LIN {X 0,Y 217.024,Z 808.035,A -85,B 0,C 180,E1 -22006.463,E2 -22006.463} C_VEL
LIN {X 0,Y 209.804,Z 820.642,A -85,B 0,C 180,E1 -22009.848,E2 -22009.848} C_VEL
LIN {X 0,Y 205.023,Z 828.704,A -85,B 0,C 180,E1 -22012.523,E2 -22012.523} C_VEL
LIN {X 0,Y 199.918,Z 836.875,A -85,B 0,C 180,E1 -22015.774,E2 -22015.774} C_VEL
LIN {X 0,Y 196.083,Z 843.017,A -85,B 0,C 180,E1 -22018.688,E2 -22018.688} C_VEL
LIN {X 0,Y 191.79,Z 849.969,A -85,B 0,C 180,E1 -22022.739,E2 -22022.739} C_VEL
LIN {X 0,Y 188.385,Z 855.734,A -85,B 0,C 180,E1 -22026.939,E2 -22026.939} C_VEL
LIN {X 0,Y 186.27,Z 859.773,A -85,B 0,C 180,E1 -22030.606,E2 -22030.606} C_VEL
LIN {X 0,Y 184.562,Z 863.22,A -85,B 0,C 180,E1 -22034.541,E2 -22034.541} C_VEL
LIN {X 0,Y 183.409,Z 866.084,A -85,B 0,C 180,E1 -22038.954,E2 -22038.954} C_VEL
LIN {X 0,Y 183.157,Z 867.229,A -85,B 0,C 180,E1 -22041.171,E2 -22041.171} C_VEL
LIN {X 0,Y 183.027,Z 868.67,A -85,B 0,C 180,E1 -22045.596,E2 -22045.596} C_VEL
LIN {X 0,Y 183.139,Z 869.152,A -85,B 0,C 180,E1 -22050,E2 -22050} C_VEL
LIN {X 0,Y 183.027,Z 868.67,A -85,B 0,C 180,E1 -22054.404,E2 -22054.404} C_VEL
LIN {X 0,Y 183.156,Z 867.229,A -85,B 0,C 180,E1 -22058.829,E2 -22058.829} C_VEL
LIN {X 0,Y 183.829,Z 864.826,A -85,B 0,C 180,E1 -22063.261,E2 -22063.261} C_VEL
LIN {X 0,Y 185.438,Z 861.443,A -85,B 0,C 180,E1 -22067.649,E2 -22067.649} C_VEL
LIN {X 0,Y 187.698,Z 857.024,A -85,B 0,C 180,E1 -22071.989,E2 -22071.989} C_VEL
LIN {X 0,Y 190.882,Z 851.516,A -85,B 0,C 180,E1 -22076.22,E2 -22076.22} C_VEL
LIN {X 0,Y 194.222,Z 845.918,A -85,B 0,C 180,E1 -22079.721,E2 -22079.721} C_VEL
LIN {X 0,Y 198.584,Z 838.981,A -85,B 0,C 180,E1 -22083.267,E2 -22083.267} C_VEL
LIN {X 0,Y 202.834,Z 832.332,A -85,B 0,C 180,E1 -22086.087,E2 -22086.087} C_VEL
LIN {X 0,Y 207.695,Z 824.178,A -85,B 0,C 180,E1 -22089.026,E2 -22089.026} C_VEL
LIN {X 0,Y 212.368,Z 816.196,A -85,B 0,C 180,E1 -22091.441,E2 -22091.441} C_VEL
LIN {X 0,Y 217.847,Z 806.411,A -85,B 0,C 180,E1 -22093.916,E2 -22093.916} C_VEL
LIN {X 0,Y 223.353,Z 796.062,A -85,B 0,C 180,E1 -22096.079,E2 -22096.079} C_VEL
LIN {X 0,Y 228.421,Z 785.635,A -85,B 0,C 180,E1 -22097.924,E2 -22097.924} C_VEL
LIN {X 0,Y 233.261,Z 774.829,A -85,B 0,C 180,E1 -22099.53,E2 -22099.53} C_VEL
LIN {X 0,Y 237.755,Z 763.897,A -85,B 0,C 180,E1 -22100.889,E2 -22100.889} C_VEL
LIN {X 0,Y 242.076,Z 752.106,A -85,B 0,C 180,E1 -22102.121,E2 -22102.121} C_VEL
LIN {X 0,Y 246.197,Z 739.235,A -85,B 0,C 180,E1 -22103.231,E2 -22103.231} C_VEL
LIN {X 0,Y 249.836,Z 726.035,A -85,B 0,C 180,E1 -22104.144,E2 -22104.144} C_VEL
LIN {X 0,Y 252.794,Z 713.298,A -85,B 0,C 180,E1 -22104.836,E2 -22104.836} C_VEL
LIN {X 0,Y 255.143,Z 700.698,A -85,B 0,C 180,E1 -22105.376,E2 -22105.376} C_VEL
LIN {X 0,Y 256.972,Z 687.246,A -85,B 0,C 180,E1 -22105.822,E2 -22105.822} C_VEL
LIN {X 0,Y 259.606,Z 655.333,A -85,B 0,C 180,E1 -22106.613,E2 -22106.613} C_VEL
LIN {X 0,Y 264.674,Z 589.177,A -85,B 0,C 180,E1 -22108.172,E2 -22108.172} C_VEL
LIN {X 0,Y 260.374,Z 578.709,A -85,B 0,C 180,E1 -22110.28,E2 -22110.28} C_VEL
LIN {X 0,Y 255.377,Z 567.773,A -85,B 0,C 180,E1 -22112.939,E2 -22112.939} C_VEL
LIN {X 0,Y 251.472,Z 560.216,A -85,B 0,C 180,E1 -22115.215,E2 -22115.215} C_VEL
LIN {X 0,Y 247.589,Z 554.194,A -85,B 0,C 180,E1 -22117.66,E2 -22117.66} C_VEL
LIN {X 0,Y 245.205,Z 550.628,A -85,B 0,C 180,E1 -22119.327,E2 -22119.327} C_VEL
LIN {X 0,Y 242.508,Z 546.779,A -85,B 0,C 180,E1 -22121.41,E2 -22121.41} C_VEL
LIN {X 0,Y 239.491,Z 542.43,A -85,B 0,C 180,E1 -22124.116,E2 -22124.116} C_VEL
LIN {X 0,Y 237.073,Z 538.972,A -85,B 0,C 180,E1 -22126.718,E2 -22126.718} C_VEL
LIN {X 0,Y 236.559,Z 538.249,A -85,B 0,C 180,E1 -22127.343,E2 -22127.343} C_VEL
LIN {X 0,Y 234.058,Z 535.194,A -85,B 0,C 180,E1 -22130.93,E2 -22130.93} C_VEL
LIN {X 0,Y 233.366,Z 533.383,A -85,B 0,C 180,E1 -22132.429,E2 -22132.429} C_VEL
LIN {X 0,Y 231.434,Z 531.641,A -85,B 0,C 180,E1 -22140,E2 -22140} C_VEL
LIN {X 0,Y 233.419,Z 533.525,A -85,B 0,C 180,E1 -22148.113,E2 -22148.113} C_VEL
LIN {X 0,Y 235.107,Z 536.867,A -85,B 0,C 180,E1 -22151.204,E2 -22151.204} C_VEL
LIN {X 0,Y 237.005,Z 538.845,A -85,B 0,C 180,E1 -22153.613,E2 -22153.613} C_VEL
LIN {X 0,Y 239.475,Z 542.534,A -85,B 0,C 180,E1 -22156.298,E2 -22156.298} C_VEL
LIN {X 0,Y 240.592,Z 544.125,A -85,B 0,C 180,E1 -22157.353,E2 -22157.353} C_VEL
LIN {X 0,Y 243.915,Z 548.714,A -85,B 0,C 180,E1 -22160.118,E2 -22160.118} C_VEL
LIN {X 0,Y 246.909,Z 553.171,A -85,B 0,C 180,E1 -22162.296,E2 -22162.296} C_VEL
LIN {X 0,Y 251.503,Z 560.18,A -85,B 0,C 180,E1 -22165.214,E2 -22165.214} C_VEL
LIN {X 0,Y 256.264,Z 567.994,A -85,B 0,C 180,E1 -22167.872,E2 -22167.872} C_VEL
LIN {X 0,Y 263.831,Z 578.938,A -85,B 0,C 180,E1 -22171.427,E2 -22171.427} C_VEL
LIN {X 0,Y 270.208,Z 586.445,A -85,B 0,C 180,E1 -22173.945,E2 -22173.945} C_VEL
LIN {X 0,Y 277.709,Z 593.975,A -85,B 0,C 180,E1 -22176.52,E2 -22176.52} C_VEL
LIN {X 0,Y 287.772,Z 602.451,A -85,B 0,C 180,E1 -22179.509,E2 -22179.509} C_VEL
LIN {X 0,Y 295.037,Z 608.473,A -85,B 0,C 180,E1 -22181.667,E2 -22181.667} C_VEL
LIN {X 0,Y 301.973,Z 614.367,A -85,B 0,C 180,E1 -22183.92,E2 -22183.92} C_VEL
LIN {X 0,Y 307.887,Z 619.394,A -85,B 0,C 180,E1 -22185.977,E2 -22185.977} C_VEL
LIN {X 0,Y 314.535,Z 625.112,A -85,B 0,C 180,E1 -22188.552,E2 -22188.552} C_VEL
LIN {X 0,Y 320.194,Z 630.065,A -85,B 0,C 180,E1 -22190.886,E2 -22190.886} C_VEL
LIN {X 0,Y 327.166,Z 636.13,A -85,B 0,C 180,E1 -22193.896,E2 -22193.896} C_VEL
LIN {X 0,Y 331.947,Z 639.962,A -85,B 0,C 180,E1 -22196.053,E2 -22196.053} C_VEL
LIN {X 0,Y 336.603,Z 643.968,A -85,B 0,C 180,E1 -22198.269,E2 -22198.269} C_VEL
LIN {X 0,Y 340.503,Z 647.021,A -85,B 0,C 180,E1 -22200.202,E2 -22200.202} C_VEL
LIN {X 0,Y 344.944,Z 651.021,A -85,B 0,C 180,E1 -22202.581,E2 -22202.581} C_VEL
LIN {X 0,Y 349.886,Z 654.477,A -85,B 0,C 180,E1 -22205.377,E2 -22205.377} C_VEL
LIN {X 0,Y 353.537,Z 657.803,A -85,B 0,C 180,E1 -22207.688,E2 -22207.688} C_VEL
LIN {X 0,Y 357.378,Z 660.485,A -85,B 0,C 180,E1 -22210.301,E2 -22210.301} C_VEL
LIN {X 0,Y 359.995,Z 662.174,A -85,B 0,C 180,E1 -22212.302,E2 -22212.302} C_VEL
LIN {X 0,Y 362.803,Z 664.895,A -85,B 0,C 180,E1 -22214.773,E2 -22214.773} C_VEL
LIN {X 0,Y 365.298,Z 666.919,A -85,B 0,C 180,E1 -22217.353,E2 -22217.353} C_VEL
LIN {X 0,Y 367.182,Z 668.028,A -85,B 0,C 180,E1 -22219.57,E2 -22219.57} C_VEL
LIN {X 0,Y 369.013,Z 668.858,A -85,B 0,C 180,E1 -22222.339,E2 -22222.339} C_VEL
LIN {X 0,Y 370.309,Z 669.612,A -85,B 0,C 180,E1 -22225.096,E2 -22225.096} C_VEL
LIN {X 0,Y 371.028,Z 669.847,A -85,B 0,C 180,E1 -22227.829,E2 -22227.829} C_VEL
LIN {X 0,Y 371.228,Z 669.986,A -85,B 0,C 180,E1 -22230,E2 -22230} C_VEL
LIN {X 0,Y 371.028,Z 669.845,A -85,B 0,C 180,E1 -22232.171,E2 -22232.171} C_VEL
LIN {X 0,Y 370.309,Z 669.617,A -85,B 0,C 180,E1 -22234.904,E2 -22234.904} C_VEL
LIN {X 0,Y 369.013,Z 668.859,A -85,B 0,C 180,E1 -22237.661,E2 -22237.661} C_VEL
LIN {X 0,Y 367.28,Z 668.119,A -85,B 0,C 180,E1 -22240.312,E2 -22240.312} C_VEL
LIN {X 0,Y 364.987,Z 666.71,A -85,B 0,C 180,E1 -22243,E2 -22243} C_VEL
LIN {X 0,Y 362.396,Z 664.592,A -85,B 0,C 180,E1 -22245.579,E2 -22245.579} C_VEL
LIN {X 0,Y 359.357,Z 661.588,A -85,B 0,C 180,E1 -22248.235,E2 -22248.235} C_VEL
LIN {X 0,Y 356.069,Z 659.663,A -85,B 0,C 180,E1 -22250.596,E2 -22250.596} C_VEL
LIN {X 0,Y 352.093,Z 656.652,A -85,B 0,C 180,E1 -22253.233,E2 -22253.233} C_VEL
LIN {X 0,Y 348.854,Z 653.633,A -85,B 0,C 180,E1 -22255.248,E2 -22255.248} C_VEL
LIN {X 0,Y 344.683,Z 650.803,A -85,B 0,C 180,E1 -22257.562,E2 -22257.562} C_VEL
LIN {X 0,Y 339.913,Z 646.465,A -85,B 0,C 180,E1 -22260.097,E2 -22260.097} C_VEL
LIN {X 0,Y 334.266,Z 642.131,A -85,B 0,C 180,E1 -22262.846,E2 -22262.846} C_VEL
LIN {X 0,Y 329.785,Z 638.132,A -85,B 0,C 180,E1 -22264.941,E2 -22264.941} C_VEL
LIN {X 0,Y 324.302,Z 633.671,A -85,B 0,C 180,E1 -22267.357,E2 -22267.357} C_VEL
LIN {X 0,Y 319.804,Z 629.722,A -85,B 0,C 180,E1 -22269.277,E2 -22269.277} C_VEL
LIN {X 0,Y 314.166,Z 624.78,A -85,B 0,C 180,E1 -22271.598,E2 -22271.598} C_VEL
LIN {X 0,Y 307.596,Z 619.166,A -85,B 0,C 180,E1 -22274.126,E2 -22274.126} C_VEL
LIN {X 0,Y 301.98,Z 614.344,A -85,B 0,C 180,E1 -22276.079,E2 -22276.079} C_VEL
LIN {X 0,Y 295.594,Z 608.892,A -85,B 0,C 180,E1 -22278.155,E2 -22278.155} C_VEL
LIN {X 0,Y 288.716,Z 603.223,A -85,B 0,C 180,E1 -22280.223,E2 -22280.223} C_VEL
LIN {X 0,Y 279.821,Z 595.822,A -85,B 0,C 180,E1 -22282.818,E2 -22282.818} C_VEL
LIN {X 0,Y 271.936,Z 588.351,A -85,B 0,C 180,E1 -22285.426,E2 -22285.426} C_VEL
LIN {X 0,Y 264.195,Z 579.408,A -85,B 0,C 180,E1 -22288.419,E2 -22288.419} C_VEL
LIN {X 0,Y 256.457,Z 568.307,A -85,B 0,C 180,E1 -22292.027,E2 -22292.027} C_VEL
LIN {X 0,Y 251.912,Z 560.875,A -85,B 0,C 180,E1 -22294.542,E2 -22294.542} C_VEL
LIN {X 0,Y 247.439,Z 553.984,A -85,B 0,C 180,E1 -22297.343,E2 -22297.343} C_VEL
LIN {X 0,Y 244.959,Z 550.237,A -85,B 0,C 180,E1 -22299.094,E2 -22299.094} C_VEL
LIN {X 0,Y 242.778,Z 547.152,A -85,B 0,C 180,E1 -22300.775,E2 -22300.775} C_VEL
LIN {X 0,Y 239.641,Z 542.684,A -85,B 0,C 180,E1 -22303.55,E2 -22303.55} C_VEL
LIN {X 0,Y 237.165,Z 539.221,A -85,B 0,C 180,E1 -22306.178,E2 -22306.178} C_VEL
LIN {X 0,Y 236.484,Z 538.21,A -85,B 0,C 180,E1 -22307.012,E2 -22307.012} C_VEL
LIN {X 0,Y 234.186,Z 535.427,A -85,B 0,C 180,E1 -22310.282,E2 -22310.282} C_VEL
LIN {X 0,Y 233.268,Z 533.307,A -85,B 0,C 180,E1 -22312.208,E2 -22312.208} C_VEL
LIN {X 0,Y 231.434,Z 531.64,A -85,B 0,C 180,E1 -22320,E2 -22320} C_VEL
LIN {X 0,Y 233.413,Z 533.486,A -85,B 0,C 180,E1 -22327.679,E2 -22327.679} C_VEL
LIN {X 0,Y 235.097,Z 536.825,A -85,B 0,C 180,E1 -22330.769,E2 -22330.769} C_VEL
LIN {X 0,Y 236.992,Z 538.793,A -85,B 0,C 180,E1 -22333.178,E2 -22333.178} C_VEL
LIN {X 0,Y 239.142,Z 542.101,A -85,B 0,C 180,E1 -22335.556,E2 -22335.556} C_VEL
LIN {X 0,Y 240.394,Z 543.725,A -85,B 0,C 180,E1 -22336.744,E2 -22336.744} C_VEL
LIN {X 0,Y 243.948,Z 548.807,A -85,B 0,C 180,E1 -22339.732,E2 -22339.732} C_VEL
LIN {X 0,Y 246.984,Z 553.277,A -85,B 0,C 180,E1 -22341.93,E2 -22341.93} C_VEL
LIN {X 0,Y 251.076,Z 559.526,A -85,B 0,C 180,E1 -22344.544,E2 -22344.544} C_VEL
LIN {X 0,Y 254.166,Z 565.218,A -85,B 0,C 180,E1 -22346.369,E2 -22346.369} C_VEL
LIN {X 0,Y 259.878,Z 577.475,A -85,B 0,C 180,E1 -22349.463,E2 -22349.463} C_VEL
LIN {X 0,Y 264.683,Z 589.177,A -85,B 0,C 180,E1 -22351.831,E2 -22351.831} C_VEL
LIN {X 0,Y 257.13,Z 685.944,A -85,B 0,C 180,E1 -22354.143,E2 -22354.143} C_VEL
LIN {X 0,Y 255.437,Z 698.699,A -85,B 0,C 180,E1 -22354.546,E2 -22354.546} C_VEL
LIN {X 0,Y 253.09,Z 711.765,A -85,B 0,C 180,E1 -22355.086,E2 -22355.086} C_VEL
LIN {X 0,Y 250.427,Z 723.566,A -85,B 0,C 180,E1 -22355.7,E2 -22355.7} C_VEL
LIN {X 0,Y 247.095,Z 736.159,A -85,B 0,C 180,E1 -22356.536,E2 -22356.536} C_VEL
LIN {X 0,Y 243.326,Z 748.397,A -85,B 0,C 180,E1 -22357.538,E2 -22357.538} C_VEL
LIN {X 0,Y 238.912,Z 760.899,A -85,B 0,C 180,E1 -22358.783,E2 -22358.783} C_VEL
LIN {X 0,Y 234.406,Z 772.222,A -85,B 0,C 180,E1 -22360.135,E2 -22360.135} C_VEL
LIN {X 0,Y 229.479,Z 783.349,A -85,B 0,C 180,E1 -22361.713,E2 -22361.713} C_VEL
LIN {X 0,Y 224.821,Z 793.183,A -85,B 0,C 180,E1 -22363.384,E2 -22363.384} C_VEL
LIN {X 0,Y 219.863,Z 802.865,A -85,B 0,C 180,E1 -22365.314,E2 -22365.314} C_VEL
LIN {X 0,Y 217.024,Z 808.035,A -85,B 0,C 180,E1 -22366.463,E2 -22366.463} C_VEL
LIN {X 0,Y 214.287,Z 812.154,A -85,B 0,C 180,E1 -22367.329,E2 -22367.329} C_VEL
LIN {X 0,Y 208.286,Z 818.645,A -85,B 0,C 180,E1 -22368.566,E2 -22368.566} C_VEL
LIN {X 0,Y 202.265,Z 824.691,A -85,B 0,C 180,E1 -22369.975,E2 -22369.975} C_VEL
LIN {X 0,Y 199.551,Z 828.11,A -85,B 0,C 180,E1 -22371.106,E2 -22371.106} C_VEL
LIN {X 0,Y 193.984,Z 836.662,A -85,B 0,C 180,E1 -22374.573,E2 -22374.573} C_VEL
LIN {X 0,Y 189.938,Z 842.803,A -85,B 0,C 180,E1 -22377.554,E2 -22377.554} C_VEL
LIN {X 0,Y 185.391,Z 849.755,A -85,B 0,C 180,E1 -22381.715,E2 -22381.715} C_VEL
LIN {X 0,Y 181.771,Z 855.521,A -85,B 0,C 180,E1 -22386.049,E2 -22386.049} C_VEL
LIN {X 0,Y 179.735,Z 859.145,A -85,B 0,C 180,E1 -22389.396,E2 -22389.396} C_VEL
LIN {X 0,Y 177.65,Z 863.008,A -85,B 0,C 180,E1 -22393.924,E2 -22393.924} C_VEL
LIN {X 0,Y 176.388,Z 865.873,A -85,B 0,C 180,E1 -22398.509,E2 -22398.509} C_VEL
LIN {X 0,Y 176.08,Z 867.017,A -85,B 0,C 180,E1 -22400.813,E2 -22400.813} C_VEL
LIN {X 0,Y 175.936,Z 868.459,A -85,B 0,C 180,E1 -22405.418,E2 -22405.418} C_VEL
LIN {X 0,Y 176.048,Z 868.943,A -85,B 0,C 180,E1 -22410,E2 -22410} C_VEL
LIN {X 0,Y 175.936,Z 868.459,A -85,B 0,C 180,E1 -22414.582,E2 -22414.582} C_VEL
LIN {X 0,Y 176.079,Z 867.017,A -85,B 0,C 180,E1 -22419.187,E2 -22419.187} C_VEL
LIN {X 0,Y 176.855,Z 864.614,A -85,B 0,C 180,E1 -22423.794,E2 -22423.794} C_VEL
LIN {X 0,Y 179.323,Z 859.848,A -85,B 0,C 180,E1 -22429.847,E2 -22429.847} C_VEL
LIN {X 0,Y 181.033,Z 856.811,A -85,B 0,C 180,E1 -22432.843,E2 -22432.843} C_VEL
LIN {X 0,Y 184.415,Z 851.302,A -85,B 0,C 180,E1 -22437.213,E2 -22437.213} C_VEL
LIN {X 0,Y 187.644,Z 846.219,A -85,B 0,C 180,E1 -22440.521,E2 -22440.521} C_VEL
LIN {X 0,Y 192.602,Z 838.768,A -85,B 0,C 180,E1 -22444.442,E2 -22444.442} C_VEL
LIN {X 0,Y 197.05,Z 832.119,A -85,B 0,C 180,E1 -22447.323,E2 -22447.323} C_VEL
LIN {X 0,Y 201.93,Z 824.313,A -85,B 0,C 180,E1 -22450.2,E2 -22450.2} C_VEL
LIN {X 0,Y 207.021,Z 815.983,A -85,B 0,C 180,E1 -22452.761,E2 -22452.761} C_VEL
LIN {X 0,Y 212.732,Z 806.198,A -85,B 0,C 180,E1 -22455.257,E2 -22455.257} C_VEL
LIN {X 0,Y 217.992,Z 796.721,A -85,B 0,C 180,E1 -22457.266,E2 -22457.266} C_VEL
LIN {X 0,Y 223.141,Z 786.567,A -85,B 0,C 180,E1 -22459.102,E2 -22459.102} C_VEL
LIN {X 0,Y 228.685,Z 774.618,A -85,B 0,C 180,E1 -22460.893,E2 -22460.893} C_VEL
LIN {X 0,Y 233.303,Z 763.685,A -85,B 0,C 180,E1 -22462.254,E2 -22462.254} C_VEL
LIN {X 0,Y 237.693,Z 752.113,A -85,B 0,C 180,E1 -22463.457,E2 -22463.457} C_VEL
LIN {X 0,Y 241.996,Z 739.024,A -85,B 0,C 180,E1 -22464.584,E2 -22464.584} C_VEL
LIN {X 0,Y 245.739,Z 725.825,A -85,B 0,C 180,E1 -22465.487,E2 -22465.487} C_VEL
LIN {X 0,Y 248.78,Z 713.088,A -85,B 0,C 180,E1 -22466.171,E2 -22466.171} C_VEL
LIN {X 0,Y 251.178,Z 700.488,A -85,B 0,C 180,E1 -22466.708,E2 -22466.708} C_VEL
LIN {X 0,Y 253.054,Z 687.036,A -85,B 0,C 180,E1 -22467.151,E2 -22467.151} C_VEL
LIN {X 0,Y 255.611,Z 656.913,A -85,B 0,C 180,E1 -22467.905,E2 -22467.905} C_VEL
LIN {X 0,Y 260.741,Z 592.077,A -85,B 0,C 180,E1 -22469.427,E2 -22469.427} C_VEL
LIN {X 0,Y 256.898,Z 582.594,A -85,B 0,C 180,E1 -22471.433,E2 -22471.433} C_VEL
LIN {X 0,Y 252.212,Z 572.078,A -85,B 0,C 180,E1 -22474.095,E2 -22474.095} C_VEL
LIN {X 0,Y 249.051,Z 565.842,A -85,B 0,C 180,E1 -22476.047,E2 -22476.047} C_VEL
LIN {X 0,Y 244.194,Z 558.051,A -85,B 0,C 180,E1 -22479.349,E2 -22479.349} C_VEL
LIN {X 0,Y 240.903,Z 553.362,A -85,B 0,C 180,E1 -22481.942,E2 -22481.942} C_VEL
LIN {X 0,Y 238.071,Z 549.141,A -85,B 0,C 180,E1 -22484.592,E2 -22484.592} C_VEL
LIN {X 0,Y 235.63,Z 545.389,A -85,B 0,C 180,E1 -22487.375,E2 -22487.375} C_VEL
LIN {X 0,Y 232.899,Z 541.908,A -85,B 0,C 180,E1 -22491.431,E2 -22491.431} C_VEL
LIN {X 0,Y 232.289,Z 540.323,A -85,B 0,C 180,E1 -22492.83,E2 -22492.83} C_VEL
LIN {X 0,Y 230.568,Z 538.691,A -85,B 0,C 180,E1 -22500,E2 -22500} C_VEL
LIN {X 0,Y 232.394,Z 540.489,A -85,B 0,C 180,E1 -22507.821,E2 -22507.821} C_VEL
LIN {X 0,Y 234.094,Z 543.891,A -85,B 0,C 180,E1 -22511.034,E2 -22511.034} C_VEL
LIN {X 0,Y 235.74,Z 545.661,A -85,B 0,C 180,E1 -22513.194,E2 -22513.194} C_VEL
LIN {X 0,Y 238.295,Z 549.47,A -85,B 0,C 180,E1 -22516.051,E2 -22516.051} C_VEL
LIN {X 0,Y 242.459,Z 555.551,A -85,B 0,C 180,E1 -22519.747,E2 -22519.747} C_VEL
LIN {X 0,Y 245.212,Z 559.806,A -85,B 0,C 180,E1 -22521.82,E2 -22521.82} C_VEL
LIN {X 0,Y 249.252,Z 566.131,A -85,B 0,C 180,E1 -22524.492,E2 -22524.492} C_VEL
LIN {X 0,Y 253.711,Z 573.674,A -85,B 0,C 180,E1 -22527.102,E2 -22527.102} C_VEL
LIN {X 0,Y 261.405,Z 585.093,A -85,B 0,C 180,E1 -22530.865,E2 -22530.865} C_VEL
LIN {X 0,Y 267.642,Z 592.574,A -85,B 0,C 180,E1 -22533.409,E2 -22533.409} C_VEL
LIN {X 0,Y 275.276,Z 600.336,A -85,B 0,C 180,E1 -22536.103,E2 -22536.103} C_VEL
LIN {X 0,Y 289.9,Z 612.757,A -85,B 0,C 180,E1 -22540.475,E2 -22540.475} C_VEL
LIN {X 0,Y 296.185,Z 617.8,A -85,B 0,C 180,E1 -22542.391,E2 -22542.391} C_VEL
LIN {X 0,Y 302.458,Z 622.865,A -85,B 0,C 180,E1 -22544.429,E2 -22544.429} C_VEL
LIN {X 0,Y 308.854,Z 628.471,A -85,B 0,C 180,E1 -22546.732,E2 -22546.732} C_VEL
LIN {X 0,Y 313.492,Z 632.478,A -85,B 0,C 180,E1 -22548.54,E2 -22548.54} C_VEL
LIN {X 0,Y 319.336,Z 637.404,A -85,B 0,C 180,E1 -22550.94,E2 -22550.94} C_VEL
LIN {X 0,Y 325.614,Z 642.904,A -85,B 0,C 180,E1 -22553.642,E2 -22553.642} C_VEL
LIN {X 0,Y 330.476,Z 646.77,A -85,B 0,C 180,E1 -22555.815,E2 -22555.815} C_VEL
LIN {X 0,Y 335.102,Z 650.715,A -85,B 0,C 180,E1 -22557.99,E2 -22557.99} C_VEL
LIN {X 0,Y 338.902,Z 653.671,A -85,B 0,C 180,E1 -22559.871,E2 -22559.871} C_VEL
LIN {X 0,Y 343.55,Z 657.813,A -85,B 0,C 180,E1 -22562.326,E2 -22562.326} C_VEL
LIN {X 0,Y 348.565,Z 661.301,A -85,B 0,C 180,E1 -22565.136,E2 -22565.136} C_VEL
LIN {X 0,Y 352.247,Z 664.636,A -85,B 0,C 180,E1 -22567.427,E2 -22567.427} C_VEL
LIN {X 0,Y 356.173,Z 667.387,A -85,B 0,C 180,E1 -22570.095,E2 -22570.095} C_VEL
LIN {X 0,Y 358.955,Z 669.162,A -85,B 0,C 180,E1 -22572.175,E2 -22572.175} C_VEL
LIN {X 0,Y 361.661,Z 671.815,A -85,B 0,C 180,E1 -22574.557,E2 -22574.557} C_VEL
LIN {X 0,Y 364.213,Z 673.832,A -85,B 0,C 180,E1 -22577.117,E2 -22577.117} C_VEL
LIN {X 0,Y 366.284,Z 675.068,A -85,B 0,C 180,E1 -22579.544,E2 -22579.544} C_VEL
LIN {X 0,Y 368.135,Z 675.877,A -85,B 0,C 180,E1 -22582.32,E2 -22582.32} C_VEL
LIN {X 0,Y 369.44,Z 676.657,A -85,B 0,C 180,E1 -22585.084,E2 -22585.084} C_VEL
LIN {X 0,Y 370.159,Z 676.892,A -85,B 0,C 180,E1 -22587.824,E2 -22587.824} C_VEL
LIN {X 0,Y 370.363,Z 677.032,A -85,B 0,C 180,E1 -22590,E2 -22590} C_VEL
LIN {X 0,Y 370.159,Z 676.891,A -85,B 0,C 180,E1 -22592.176,E2 -22592.176} C_VEL
LIN {X 0,Y 369.439,Z 676.663,A -85,B 0,C 180,E1 -22594.915,E2 -22594.915} C_VEL
LIN {X 0,Y 368.134,Z 675.885,A -85,B 0,C 180,E1 -22597.68,E2 -22597.68} C_VEL
LIN {X 0,Y 366.382,Z 675.159,A -85,B 0,C 180,E1 -22600.338,E2 -22600.338} C_VEL
LIN {X 0,Y 364.085,Z 673.731,A -85,B 0,C 180,E1 -22603.033,E2 -22603.033} C_VEL
LIN {X 0,Y 361.459,Z 671.656,A -85,B 0,C 180,E1 -22605.62,E2 -22605.62} C_VEL
LIN {X 0,Y 358.395,Z 668.607,A -85,B 0,C 180,E1 -22608.285,E2 -22608.285} C_VEL
LIN {X 0,Y 355.091,Z 666.685,A -85,B 0,C 180,E1 -22610.656,E2 -22610.656} C_VEL
LIN {X 0,Y 351.069,Z 663.714,A -85,B 0,C 180,E1 -22613.303,E2 -22613.303} C_VEL
LIN {X 0,Y 347.314,Z 660.308,A -85,B 0,C 180,E1 -22615.608,E2 -22615.608} C_VEL
LIN {X 0,Y 343.32,Z 657.597,A -85,B 0,C 180,E1 -22617.803,E2 -22617.803} C_VEL
LIN {X 0,Y 338.616,Z 653.421,A -85,B 0,C 180,E1 -22620.274,E2 -22620.274} C_VEL
LIN {X 0,Y 332.904,Z 649.018,A -85,B 0,C 180,E1 -22623.043,E2 -22623.043} C_VEL
LIN {X 0,Y 327.743,Z 644.483,A -85,B 0,C 180,E1 -22625.428,E2 -22625.428} C_VEL
LIN {X 0,Y 322.376,Z 640.13,A -85,B 0,C 180,E1 -22627.769,E2 -22627.769} C_VEL
LIN {X 0,Y 317.673,Z 636.043,A -85,B 0,C 180,E1 -22629.749,E2 -22629.749} C_VEL
LIN {X 0,Y 312.278,Z 631.353,A -85,B 0,C 180,E1 -22631.947,E2 -22631.947} C_VEL
LIN {X 0,Y 305.786,Z 625.92,A -85,B 0,C 180,E1 -22634.382,E2 -22634.382} C_VEL
LIN {X 0,Y 300.757,Z 621.582,A -85,B 0,C 180,E1 -22636.124,E2 -22636.124} C_VEL
LIN {X 0,Y 294.652,Z 616.46,A -85,B 0,C 180,E1 -22638.099,E2 -22638.099} C_VEL
LIN {X 0,Y 286.82,Z 610.155,A -85,B 0,C 180,E1 -22640.426,E2 -22640.426} C_VEL
LIN {X 0,Y 276.881,Z 601.705,A -85,B 0,C 180,E1 -22643.381,E2 -22643.381} C_VEL
LIN {X 0,Y 269.548,Z 594.713,A -85,B 0,C 180,E1 -22645.877,E2 -22645.877} C_VEL
LIN {X 0,Y 261.638,Z 585.413,A -85,B 0,C 180,E1 -22649.032,E2 -22649.032} C_VEL
LIN {X 0,Y 253.855,Z 573.918,A -85,B 0,C 180,E1 -22652.82,E2 -22652.82} C_VEL
LIN {X 0,Y 248.762,Z 565.295,A -85,B 0,C 180,E1 -22655.818,E2 -22655.818} C_VEL
LIN {X 0,Y 243.681,Z 557.331,A -85,B 0,C 180,E1 -22659.311,E2 -22659.311} C_VEL
LIN {X 0,Y 241.172,Z 553.688,A -85,B 0,C 180,E1 -22661.304,E2 -22661.304} C_VEL
LIN {X 0,Y 238.084,Z 549.235,A -85,B 0,C 180,E1 -22664.155,E2 -22664.155} C_VEL
LIN {X 0,Y 235.68,Z 545.544,A -85,B 0,C 180,E1 -22666.885,E2 -22666.885} C_VEL
LIN {X 0,Y 233.021,Z 542.13,A -85,B 0,C 180,E1 -22670.78,E2 -22670.78} C_VEL
LIN {X 0,Y 232.196,Z 540.262,A -85,B 0,C 180,E1 -22672.61,E2 -22672.61} C_VEL
LIN {X 0,Y 230.568,Z 538.689,A -85,B 0,C 180,E1 -22680,E2 -22680} C_VEL
LIN {X 0,Y 232.418,Z 540.568,A -85,B 0,C 180,E1 -22687.466,E2 -22687.466} C_VEL
LIN {X 0,Y 234.156,Z 543.929,A -85,B 0,C 180,E1 -22690.703,E2 -22690.703} C_VEL
LIN {X 0,Y 235.768,Z 545.676,A -85,B 0,C 180,E1 -22692.809,E2 -22692.809} C_VEL
LIN {X 0,Y 238.175,Z 549.264,A -85,B 0,C 180,E1 -22695.511,E2 -22695.511} C_VEL
LIN {X 0,Y 242.12,Z 555.053,A -85,B 0,C 180,E1 -22699.06,E2 -22699.06} C_VEL
LIN {X 0,Y 244.964,Z 559.36,A -85,B 0,C 180,E1 -22701.222,E2 -22701.222} C_VEL
LIN {X 0,Y 249.162,Z 566.055,A -85,B 0,C 180,E1 -22704.025,E2 -22704.025} C_VEL
LIN {X 0,Y 252.103,Z 571.844,A -85,B 0,C 180,E1 -22705.84,E2 -22705.84} C_VEL
LIN {X 0,Y 257.284,Z 583.384,A -85,B 0,C 180,E1 -22708.768,E2 -22708.768} C_VEL
LIN {X 0,Y 260.754,Z 592.12,A -85,B 0,C 180,E1 -22710.579,E2 -22710.579} C_VEL
LIN {X 0,Y 253.204,Z 685.744,A -85,B 0,C 180,E1 -22712.81,E2 -22712.81} C_VEL
LIN {X 0,Y 251.316,Z 699.488,A -85,B 0,C 180,E1 -22713.249,E2 -22713.249} C_VEL
LIN {X 0,Y 248.914,Z 712.321,A -85,B 0,C 180,E1 -22713.784,E2 -22713.784} C_VEL
LIN {X 0,Y 246.034,Z 724.59,A -85,B 0,C 180,E1 -22714.432,E2 -22714.432} C_VEL
LIN {X 0,Y 242.605,Z 736.973,A -85,B 0,C 180,E1 -22715.26,E2 -22715.26} C_VEL
LIN {X 0,Y 239.2,Z 747.796,A -85,B 0,C 180,E1 -22716.152,E2 -22716.152} C_VEL
LIN {X 0,Y 235.1,Z 759.189,A -85,B 0,C 180,E1 -22717.26,E2 -22717.26} C_VEL
LIN {X 0,Y 230.424,Z 770.705,A -85,B 0,C 180,E1 -22718.597,E2 -22718.597} C_VEL
LIN {X 0,Y 225.346,Z 781.995,A -85,B 0,C 180,E1 -22720.175,E2 -22720.175} C_VEL
LIN {X 0,Y 219.961,Z 792.967,A -85,B 0,C 180,E1 -22722.026,E2 -22722.026} C_VEL
LIN {X 0,Y 214.808,Z 802.653,A -85,B 0,C 180,E1 -22723.964,E2 -22723.964} C_VEL
LIN {X 0,Y 208.882,Z 812.852,A -85,B 0,C 180,E1 -22726.392,E2 -22726.392} C_VEL
LIN {X 0,Y 203.489,Z 821.808,A -85,B 0,C 180,E1 -22728.989,E2 -22728.989} C_VEL
LIN {X 0,Y 199.551,Z 828.11,A -85,B 0,C 180,E1 -22731.106,E2 -22731.106} C_VEL
LIN {X 0,Y 196.88,Z 831.469,A -85,B 0,C 180,E1 -22732.295,E2 -22732.295} C_VEL
LIN {X 0,Y 193.446,Z 834.798,A -85,B 0,C 180,E1 -22733.363,E2 -22733.363} C_VEL
LIN {X 0,Y 185.114,Z 841.749,A -85,B 0,C 180,E1 -22735.98,E2 -22735.98} C_VEL
LIN {X 0,Y 182.584,Z 844.418,A -85,B 0,C 180,E1 -22737.401,E2 -22737.401} C_VEL
LIN {X 0,Y 179.05,Z 849.541,A -85,B 0,C 180,E1 -22740.618,E2 -22740.618} C_VEL
LIN {X 0,Y 175.191,Z 855.308,A -85,B 0,C 180,E1 -22745.089,E2 -22745.089} C_VEL
LIN {X 0,Y 172.991,Z 858.932,A -85,B 0,C 180,E1 -22748.554,E2 -22748.554} C_VEL
LIN {X 0,Y 170.745,Z 862.795,A -85,B 0,C 180,E1 -22753.255,E2 -22753.255} C_VEL
LIN {X 0,Y 169.367,Z 865.661,A -85,B 0,C 180,E1 -22758.026,E2 -22758.026} C_VEL
LIN {X 0,Y 169.027,Z 866.806,A -85,B 0,C 180,E1 -22760.426,E2 -22760.426} C_VEL
LIN {X 0,Y 168.845,Z 868.249,A -85,B 0,C 180,E1 -22765.225,E2 -22765.225} C_VEL
LIN {X 0,Y 168.959,Z 868.733,A -85,B 0,C 180,E1 -22770,E2 -22770} C_VEL
LIN {X 0,Y 168.845,Z 868.249,A -85,B 0,C 180,E1 -22774.775,E2 -22774.775} C_VEL
LIN {X 0,Y 169.025,Z 866.806,A -85,B 0,C 180,E1 -22779.574,E2 -22779.574} C_VEL
LIN {X 0,Y 169.904,Z 864.402,A -85,B 0,C 180,E1 -22784.37,E2 -22784.37} C_VEL
LIN {X 0,Y 172.371,Z 859.939,A -85,B 0,C 180,E1 -22790.319,E2 -22790.319} C_VEL
LIN {X 0,Y 174.399,Z 856.597,A -85,B 0,C 180,E1 -22793.764,E2 -22793.764} C_VEL
LIN {X 0,Y 178.017,Z 851.088,A -85,B 0,C 180,E1 -22798.277,E2 -22798.277} C_VEL
LIN {X 0,Y 181.647,Z 845.761,A -85,B 0,C 180,E1 -22801.819,E2 -22801.819} C_VEL
LIN {X 0,Y 186.703,Z 838.555,A -85,B 0,C 180,E1 -22805.693,E2 -22805.693} C_VEL
LIN {X 0,Y 191.337,Z 831.905,A -85,B 0,C 180,E1 -22808.639,E2 -22808.639} C_VEL
LIN {X 0,Y 196.32,Z 824.355,A -85,B 0,C 180,E1 -22811.471,E2 -22811.471} C_VEL
LIN {X 0,Y 201.8,Z 815.77,A -85,B 0,C 180,E1 -22814.148,E2 -22814.148} C_VEL
LIN {X 0,Y 207.75,Z 805.987,A -85,B 0,C 180,E1 -22816.661,E2 -22816.661} C_VEL
LIN {X 0,Y 212.807,Z 797.217,A -85,B 0,C 180,E1 -22818.548,E2 -22818.548} C_VEL
LIN {X 0,Y 218.504,Z 786.354,A -85,B 0,C 180,E1 -22820.527,E2 -22820.527} C_VEL
LIN {X 0,Y 224.244,Z 774.406,A -85,B 0,C 180,E1 -22822.311,E2 -22822.311} C_VEL
LIN {X 0,Y 229.011,Z 763.475,A -85,B 0,C 180,E1 -22823.664,E2 -22823.664} C_VEL
LIN {X 0,Y 233.83,Z 751.017,A -85,B 0,C 180,E1 -22824.944,E2 -22824.944} C_VEL
LIN {X 0,Y 237.931,Z 738.814,A -85,B 0,C 180,E1 -22825.985,E2 -22825.985} C_VEL
LIN {X 0,Y 241.779,Z 725.615,A -85,B 0,C 180,E1 -22826.877,E2 -22826.877} C_VEL
LIN {X 0,Y 244.903,Z 712.879,A -85,B 0,C 180,E1 -22827.549,E2 -22827.549} C_VEL
LIN {X 0,Y 247.343,Z 700.278,A -85,B 0,C 180,E1 -22828.086,E2 -22828.086} C_VEL
LIN {X 0,Y 249.26,Z 686.825,A -85,B 0,C 180,E1 -22828.527,E2 -22828.527} C_VEL
LIN {X 0,Y 252.209,Z 653.122,A -85,B 0,C 180,E1 -22829.354,E2 -22829.354} C_VEL
LIN {X 0,Y 256.922,Z 594.922,A -85,B 0,C 180,E1 -22830.73,E2 -22830.73} C_VEL
LIN {X 0,Y 252.23,Z 583.394,A -85,B 0,C 180,E1 -22833.378,E2 -22833.378} C_VEL
LIN {X 0,Y 248.359,Z 574.803,A -85,B 0,C 180,E1 -22835.783,E2 -22835.783} C_VEL
LIN {X 0,Y 246.189,Z 570.671,A -85,B 0,C 180,E1 -22837.221,E2 -22837.221} C_VEL
LIN {X 0,Y 241.853,Z 563.699,A -85,B 0,C 180,E1 -22840.367,E2 -22840.367} C_VEL
LIN {X 0,Y 239.325,Z 559.893,A -85,B 0,C 180,E1 -22842.482,E2 -22842.482} C_VEL
LIN {X 0,Y 236.768,Z 555.947,A -85,B 0,C 180,E1 -22844.973,E2 -22844.973} C_VEL
LIN {X 0,Y 234.479,Z 552.38,A -85,B 0,C 180,E1 -22847.669,E2 -22847.669} C_VEL
LIN {X 0,Y 231.714,Z 548.468,A -85,B 0,C 180,E1 -22852.045,E2 -22852.045} C_VEL
LIN {X 0,Y 231.208,Z 547.253,A -85,B 0,C 180,E1 -22853.271,E2 -22853.271} C_VEL
LIN {X 0,Y 229.704,Z 545.728,A -85,B 0,C 180,E1 -22860,E2 -22860} C_VEL
LIN {X 0,Y 231.376,Z 547.452,A -85,B 0,C 180,E1 -22867.526,E2 -22867.526} C_VEL
LIN {X 0,Y 233.085,Z 550.907,A -85,B 0,C 180,E1 -22870.862,E2 -22870.862} C_VEL
LIN {X 0,Y 234.499,Z 552.477,A -85,B 0,C 180,E1 -22872.782,E2 -22872.782} C_VEL
LIN {X 0,Y 237.51,Z 557.143,A -85,B 0,C 180,E1 -22876.215,E2 -22876.215} C_VEL
LIN {X 0,Y 241.011,Z 562.404,A -85,B 0,C 180,E1 -22879.372,E2 -22879.372} C_VEL
LIN {X 0,Y 244.673,Z 568.123,A -85,B 0,C 180,E1 -22882.148,E2 -22882.148} C_VEL
LIN {X 0,Y 249.989,Z 577.128,A -85,B 0,C 180,E1 -22885.596,E2 -22885.596} C_VEL
LIN {X 0,Y 258.341,Z 590.413,A -85,B 0,C 180,E1 -22889.991,E2 -22889.991} C_VEL
LIN {X 0,Y 265.209,Z 598.812,A -85,B 0,C 180,E1 -22892.904,E2 -22892.904} C_VEL
LIN {X 0,Y 272.726,Z 606.575,A -85,B 0,C 180,E1 -22895.635,E2 -22895.635} C_VEL
LIN {X 0,Y 288.823,Z 620.206,A -85,B 0,C 180,E1 -22900.493,E2 -22900.493} C_VEL
LIN {X 0,Y 295.573,Z 625.663,A -85,B 0,C 180,E1 -22902.552,E2 -22902.552} C_VEL
LIN {X 0,Y 302.804,Z 631.637,A -85,B 0,C 180,E1 -22904.933,E2 -22904.933} C_VEL
LIN {X 0,Y 309.037,Z 636.707,A -85,B 0,C 180,E1 -22907.188,E2 -22907.188} C_VEL
LIN {X 0,Y 315.354,Z 642.331,A -85,B 0,C 180,E1 -22909.709,E2 -22909.709} C_VEL
LIN {X 0,Y 320.561,Z 646.699,A -85,B 0,C 180,E1 -22911.883,E2 -22911.883} C_VEL
LIN {X 0,Y 326.107,Z 651.217,A -85,B 0,C 180,E1 -22914.277,E2 -22914.277} C_VEL
LIN {X 0,Y 332.445,Z 656.624,A -85,B 0,C 180,E1 -22917.195,E2 -22917.195} C_VEL
LIN {X 0,Y 337.451,Z 660.456,A -85,B 0,C 180,E1 -22919.612,E2 -22919.612} C_VEL
LIN {X 0,Y 342.214,Z 664.646,A -85,B 0,C 180,E1 -22922.099,E2 -22922.099} C_VEL
LIN {X 0,Y 346.495,Z 667.49,A -85,B 0,C 180,E1 -22924.447,E2 -22924.447} C_VEL
LIN {X 0,Y 350.858,Z 671.397,A -85,B 0,C 180,E1 -22927.133,E2 -22927.133} C_VEL
LIN {X 0,Y 354.75,Z 674.149,A -85,B 0,C 180,E1 -22929.737,E2 -22929.737} C_VEL
LIN {X 0,Y 357.912,Z 676.146,A -85,B 0,C 180,E1 -22932.049,E2 -22932.049} C_VEL
LIN {X 0,Y 360.726,Z 678.86,A -85,B 0,C 180,E1 -22934.516,E2 -22934.516} C_VEL
LIN {X 0,Y 363.306,Z 680.883,A -85,B 0,C 180,E1 -22937.085,E2 -22937.085} C_VEL
LIN {X 0,Y 365.387,Z 682.101,A -85,B 0,C 180,E1 -22939.518,E2 -22939.518} C_VEL
LIN {X 0,Y 367.253,Z 682.924,A -85,B 0,C 180,E1 -22942.302,E2 -22942.302} C_VEL
LIN {X 0,Y 368.571,Z 683.694,A -85,B 0,C 180,E1 -22945.072,E2 -22945.072} C_VEL
LIN {X 0,Y 369.291,Z 683.938,A -85,B 0,C 180,E1 -22947.819,E2 -22947.819} C_VEL
LIN {X 0,Y 369.498,Z 684.078,A -85,B 0,C 180,E1 -22950,E2 -22950} C_VEL
LIN {X 0,Y 369.291,Z 683.937,A -85,B 0,C 180,E1 -22952.181,E2 -22952.181} C_VEL
LIN {X 0,Y 368.571,Z 683.7,A -85,B 0,C 180,E1 -22954.927,E2 -22954.927} C_VEL
LIN {X 0,Y 367.253,Z 682.932,A -85,B 0,C 180,E1 -22957.698,E2 -22957.698} C_VEL
LIN {X 0,Y 365.484,Z 682.199,A -85,B 0,C 180,E1 -22960.364,E2 -22960.364} C_VEL
LIN {X 0,Y 363.18,Z 680.774,A -85,B 0,C 180,E1 -22963.066,E2 -22963.066} C_VEL
LIN {X 0,Y 360.422,Z 678.628,A -85,B 0,C 180,E1 -22965.754,E2 -22965.754} C_VEL
LIN {X 0,Y 357.216,Z 675.538,A -85,B 0,C 180,E1 -22968.488,E2 -22968.488} C_VEL
LIN {X 0,Y 353.902,Z 673.582,A -85,B 0,C 180,E1 -22970.867,E2 -22970.867} C_VEL
LIN {X 0,Y 349.933,Z 670.677,A -85,B 0,C 180,E1 -22973.444,E2 -22973.444} C_VEL
LIN {X 0,Y 345.984,Z 667.16,A -85,B 0,C 180,E1 -22975.834,E2 -22975.834} C_VEL
LIN {X 0,Y 341.882,Z 664.366,A -85,B 0,C 180,E1 -22978.086,E2 -22978.086} C_VEL
LIN {X 0,Y 336.897,Z 659.918,A -85,B 0,C 180,E1 -22980.68,E2 -22980.68} C_VEL
LIN {X 0,Y 331.16,Z 655.564,A -85,B 0,C 180,E1 -22983.416,E2 -22983.416} C_VEL
LIN {X 0,Y 326.107,Z 651.227,A -85,B 0,C 180,E1 -22985.723,E2 -22985.723} C_VEL
LIN {X 0,Y 320.206,Z 646.401,A -85,B 0,C 180,E1 -22988.268,E2 -22988.268} C_VEL
LIN {X 0,Y 315.481,Z 642.385,A -85,B 0,C 180,E1 -22990.242,E2 -22990.242} C_VEL
LIN {X 0,Y 310.053,Z 637.629,A -85,B 0,C 180,E1 -22992.409,E2 -22992.409} C_VEL
LIN {X 0,Y 303.768,Z 632.489,A -85,B 0,C 180,E1 -22994.718,E2 -22994.718} C_VEL
LIN {X 0,Y 297.454,Z 627.147,A -85,B 0,C 180,E1 -22996.867,E2 -22996.867} C_VEL
LIN {X 0,Y 289.525,Z 620.713,A -85,B 0,C 180,E1 -22999.297,E2 -22999.297} C_VEL
LIN {X 0,Y 277.423,Z 610.882,A -85,B 0,C 180,E1 -23002.841,E2 -23002.841} C_VEL
LIN {X 0,Y 266.816,Z 600.639,A -85,B 0,C 180,E1 -23006.474,E2 -23006.474} C_VEL
LIN {X 0,Y 259.112,Z 591.41,A -85,B 0,C 180,E1 -23009.658,E2 -23009.658} C_VEL
LIN {X 0,Y 251.608,Z 580.042,A -85,B 0,C 180,E1 -23013.454,E2 -23013.454} C_VEL
LIN {X 0,Y 246.768,Z 571.583,A -85,B 0,C 180,E1 -23016.425,E2 -23016.425} C_VEL
LIN {X 0,Y 241.889,Z 563.693,A -85,B 0,C 180,E1 -23019.928,E2 -23019.928} C_VEL
LIN {X 0,Y 239.399,Z 560.022,A -85,B 0,C 180,E1 -23021.999,E2 -23021.999} C_VEL
LIN {X 0,Y 236.707,Z 555.948,A -85,B 0,C 180,E1 -23024.612,E2 -23024.612} C_VEL
LIN {X 0,Y 234.17,Z 551.985,A -85,B 0,C 180,E1 -23027.653,E2 -23027.653} C_VEL
LIN {X 0,Y 231.923,Z 548.961,A -85,B 0,C 180,E1 -23031.176,E2 -23031.176} C_VEL
LIN {X 0,Y 231.332,Z 547.358,A -85,B 0,C 180,E1 -23032.582,E2 -23032.582} C_VEL
LIN {X 0,Y 229.703,Z 545.739,A -85,B 0,C 180,E1 -23040,E2 -23040} C_VEL
LIN {X 0,Y 231.367,Z 547.435,A -85,B 0,C 180,E1 -23047.089,E2 -23047.089} C_VEL
LIN {X 0,Y 233.074,Z 550.855,A -85,B 0,C 180,E1 -23050.424,E2 -23050.424} C_VEL
LIN {X 0,Y 234.555,Z 552.543,A -85,B 0,C 180,E1 -23052.437,E2 -23052.437} C_VEL
LIN {X 0,Y 236.988,Z 556.181,A -85,B 0,C 180,E1 -23055.246,E2 -23055.246} C_VEL
LIN {X 0,Y 240.923,Z 562.253,A -85,B 0,C 180,E1 -23058.882,E2 -23058.882} C_VEL
LIN {X 0,Y 244.788,Z 568.328,A -85,B 0,C 180,E1 -23061.814,E2 -23061.814} C_VEL
LIN {X 0,Y 248.005,Z 573.982,A -85,B 0,C 180,E1 -23063.979,E2 -23063.979} C_VEL
LIN {X 0,Y 252.323,Z 583.565,A -85,B 0,C 180,E1 -23066.674,E2 -23066.674} C_VEL
LIN {X 0,Y 255.991,Z 592.606,A -85,B 0,C 180,E1 -23068.768,E2 -23068.768} C_VEL
LIN {X 0,Y 256.95,Z 595.133,A -85,B 0,C 180,E1 -23069.293,E2 -23069.293} C_VEL
LIN {X 0,Y 249.431,Z 685.544,A -85,B 0,C 180,E1 -23071.44,E2 -23071.44} C_VEL
LIN {X 0,Y 247.501,Z 699.278,A -85,B 0,C 180,E1 -23071.876,E2 -23071.876} C_VEL
LIN {X 0,Y 245.021,Z 712.11,A -85,B 0,C 180,E1 -23072.398,E2 -23072.398} C_VEL
LIN {X 0,Y 242.088,Z 724.38,A -85,B 0,C 180,E1 -23073.045,E2 -23073.045} C_VEL
LIN {X 0,Y 238.583,Z 736.764,A -85,B 0,C 180,E1 -23073.87,E2 -23073.87} C_VEL
LIN {X 0,Y 234.806,Z 748.3,A -85,B 0,C 180,E1 -23074.812,E2 -23074.812} C_VEL
LIN {X 0,Y 230.841,Z 758.978,A -85,B 0,C 180,E1 -23075.847,E2 -23075.847} C_VEL
LIN {X 0,Y 226.035,Z 770.494,A -85,B 0,C 180,E1 -23077.181,E2 -23077.181} C_VEL
LIN {X 0,Y 220.787,Z 781.783,A -85,B 0,C 180,E1 -23078.753,E2 -23078.753} C_VEL
LIN {X 0,Y 215.222,Z 792.755,A -85,B 0,C 180,E1 -23080.606,E2 -23080.606} C_VEL
LIN {X 0,Y 209.887,Z 802.44,A -85,B 0,C 180,E1 -23082.554,E2 -23082.554} C_VEL
LIN {X 0,Y 203.748,Z 812.64,A -85,B 0,C 180,E1 -23085,E2 -23085} C_VEL
LIN {X 0,Y 198.085,Z 821.594,A -85,B 0,C 180,E1 -23087.616,E2 -23087.616} C_VEL
LIN {X 0,Y 192.921,Z 829.485,A -85,B 0,C 180,E1 -23090.394,E2 -23090.394} C_VEL
LIN {X 0,Y 188.156,Z 836.449,A -85,B 0,C 180,E1 -23093.301,E2 -23093.301} C_VEL
LIN {X 0,Y 183.899,Z 842.59,A -85,B 0,C 180,E1 -23096.349,E2 -23096.349} C_VEL
LIN {X 0,Y 182.584,Z 844.418,A -85,B 0,C 180,E1 -23097.401,E2 -23097.401} C_VEL
LIN {X 0,Y 180.153,Z 847.13,A -85,B 0,C 180,E1 -23098.889,E2 -23098.889} C_VEL
LIN {X 0,Y 174.719,Z 851.097,A -85,B 0,C 180,E1 -23101.239,E2 -23101.239} C_VEL
LIN {X 0,Y 169.55,Z 854.728,A -85,B 0,C 180,E1 -23103.784,E2 -23103.784} C_VEL
LIN {X 0,Y 167.589,Z 856.711,A -85,B 0,C 180,E1 -23105.546,E2 -23105.546} C_VEL
LIN {X 0,Y 164.977,Z 860.804,A -85,B 0,C 180,E1 -23110.075,E2 -23110.075} C_VEL
LIN {X 0,Y 162.984,Z 864.191,A -85,B 0,C 180,E1 -23115.006,E2 -23115.006} C_VEL
LIN {X 0,Y 161.962,Z 866.594,A -85,B 0,C 180,E1 -23120.005,E2 -23120.005} C_VEL
LIN {X 0,Y 161.736,Z 868.038,A -85,B 0,C 180,E1 -23125.014,E2 -23125.014} C_VEL
LIN {X 0,Y 161.859,Z 868.523,A -85,B 0,C 180,E1 -23130,E2 -23130} C_VEL
LIN {X 0,Y 161.736,Z 868.038,A -85,B 0,C 180,E1 -23134.986,E2 -23134.986} C_VEL
LIN {X 0,Y 161.96,Z 866.594,A -85,B 0,C 180,E1 -23139.995,E2 -23139.995} C_VEL
LIN {X 0,Y 162.975,Z 864.191,A -85,B 0,C 180,E1 -23144.995,E2 -23144.995} C_VEL
LIN {X 0,Y 165.436,Z 860.025,A -85,B 0,C 180,E1 -23150.837,E2 -23150.837} C_VEL
LIN {X 0,Y 167.803,Z 856.384,A -85,B 0,C 180,E1 -23154.76,E2 -23154.76} C_VEL
LIN {X 0,Y 171.688,Z 850.875,A -85,B 0,C 180,E1 -23159.42,E2 -23159.42} C_VEL
LIN {X 0,Y 175.385,Z 845.795,A -85,B 0,C 180,E1 -23162.911,E2 -23162.911} C_VEL
LIN {X 0,Y 180.892,Z 838.342,A -85,B 0,C 180,E1 -23167.027,E2 -23167.027} C_VEL
LIN {X 0,Y 185.752,Z 831.691,A -85,B 0,C 180,E1 -23170.03,E2 -23170.03} C_VEL
LIN {X 0,Y 190.988,Z 824.142,A -85,B 0,C 180,E1 -23172.901,E2 -23172.901} C_VEL
LIN {X 0,Y 196.703,Z 815.558,A -85,B 0,C 180,E1 -23175.607,E2 -23175.607} C_VEL
LIN {X 0,Y 201.817,Z 807.548,A -85,B 0,C 180,E1 -23177.73,E2 -23177.73} C_VEL
LIN {X 0,Y 208.562,Z 796.193,A -85,B 0,C 180,E1 -23180.189,E2 -23180.189} C_VEL
LIN {X 0,Y 214.018,Z 786.142,A -85,B 0,C 180,E1 -23182.008,E2 -23182.008} C_VEL
LIN {X 0,Y 219.936,Z 774.195,A -85,B 0,C 180,E1 -23183.788,E2 -23183.788} C_VEL
LIN {X 0,Y 224.858,Z 763.264,A -85,B 0,C 180,E1 -23185.128,E2 -23185.128} C_VEL
LIN {X 0,Y 229.311,Z 752.174,A -85,B 0,C 180,E1 -23186.275,E2 -23186.275} C_VEL
LIN {X 0,Y 233.697,Z 739.628,A -85,B 0,C 180,E1 -23187.355,E2 -23187.355} C_VEL
LIN {X 0,Y 237.633,Z 726.638,A -85,B 0,C 180,E1 -23188.24,E2 -23188.24} C_VEL
LIN {X 0,Y 241.003,Z 713.435,A -85,B 0,C 180,E1 -23188.937,E2 -23188.937} C_VEL
LIN {X 0,Y 243.654,Z 700.067,A -85,B 0,C 180,E1 -23189.508,E2 -23189.508} C_VEL
LIN {X 0,Y 245.611,Z 686.626,A -85,B 0,C 180,E1 -23189.946,E2 -23189.946} C_VEL
LIN {X 0,Y 248.825,Z 651.174,A -85,B 0,C 180,E1 -23190.796,E2 -23190.796} C_VEL
LIN {X 0,Y 253.278,Z 598.086,A -85,B 0,C 180,E1 -23192.036,E2 -23192.036} C_VEL
LIN {X 0,Y 249.172,Z 587.784,A -85,B 0,C 180,E1 -23194.516,E2 -23194.516} C_VEL
LIN {X 0,Y 245.823,Z 580.041,A -85,B 0,C 180,E1 -23196.74,E2 -23196.74} C_VEL
LIN {X 0,Y 243.631,Z 575.996,A -85,B 0,C 180,E1 -23198.268,E2 -23198.268} C_VEL
LIN {X 0,Y 240.088,Z 570.062,A -85,B 0,C 180,E1 -23200.994,E2 -23200.994} C_VEL
LIN {X 0,Y 237.634,Z 566.289,A -85,B 0,C 180,E1 -23203.148,E2 -23203.148} C_VEL
LIN {X 0,Y 235.412,Z 562.681,A -85,B 0,C 180,E1 -23205.426,E2 -23205.426} C_VEL
LIN {X 0,Y 232.965,Z 558.831,A -85,B 0,C 180,E1 -23208.471,E2 -23208.471} C_VEL
LIN {X 0,Y 230.659,Z 555.381,A -85,B 0,C 180,E1 -23212.394,E2 -23212.394} C_VEL
LIN {X 0,Y 230.181,Z 554.221,A -85,B 0,C 180,E1 -23213.617,E2 -23213.617} C_VEL
LIN {X 0,Y 228.839,Z 552.775,A -85,B 0,C 180,E1 -23220,E2 -23220} C_VEL
LIN {X 0,Y 230.362,Z 554.432,A -85,B 0,C 180,E1 -23227.229,E2 -23227.229} C_VEL
LIN {X 0,Y 232.078,Z 557.918,A -85,B 0,C 180,E1 -23230.689,E2 -23230.689} C_VEL
LIN {X 0,Y 233.289,Z 559.333,A -85,B 0,C 180,E1 -23232.394,E2 -23232.394} C_VEL
LIN {X 0,Y 236.117,Z 563.888,A -85,B 0,C 180,E1 -23235.759,E2 -23235.759} C_VEL
LIN {X 0,Y 239.397,Z 568.954,A -85,B 0,C 180,E1 -23238.84,E2 -23238.84} C_VEL
LIN {X 0,Y 242.746,Z 574.383,A -85,B 0,C 180,E1 -23241.495,E2 -23241.495} C_VEL
LIN {X 0,Y 247.333,Z 582.431,A -85,B 0,C 180,E1 -23244.634,E2 -23244.634} C_VEL
LIN {X 0,Y 256.003,Z 596.594,A -85,B 0,C 180,E1 -23249.414,E2 -23249.414} C_VEL
LIN {X 0,Y 262.692,Z 604.934,A -85,B 0,C 180,E1 -23252.348,E2 -23252.348} C_VEL
LIN {X 0,Y 270.376,Z 612.979,A -85,B 0,C 180,E1 -23255.22,E2 -23255.22} C_VEL
LIN {X 0,Y 287.033,Z 627.089,A -85,B 0,C 180,E1 -23260.302,E2 -23260.302} C_VEL
LIN {X 0,Y 295.007,Z 633.518,A -85,B 0,C 180,E1 -23262.725,E2 -23262.725} C_VEL
LIN {X 0,Y 301.848,Z 639.086,A -85,B 0,C 180,E1 -23264.971,E2 -23264.971} C_VEL
LIN {X 0,Y 308.484,Z 644.519,A -85,B 0,C 180,E1 -23267.382,E2 -23267.382} C_VEL
LIN {X 0,Y 314.277,Z 649.533,A -85,B 0,C 180,E1 -23269.676,E2 -23269.676} C_VEL
LIN {X 0,Y 319.29,Z 653.784,A -85,B 0,C 180,E1 -23271.765,E2 -23271.765} C_VEL
LIN {X 0,Y 324.928,Z 658.253,A -85,B 0,C 180,E1 -23274.187,E2 -23274.187} C_VEL
LIN {X 0,Y 331.049,Z 663.472,A -85,B 0,C 180,E1 -23276.98,E2 -23276.98} C_VEL
LIN {X 0,Y 336.145,Z 667.381,A -85,B 0,C 180,E1 -23279.424,E2 -23279.424} C_VEL
LIN {X 0,Y 340.997,Z 671.574,A -85,B 0,C 180,E1 -23281.94,E2 -23281.94} C_VEL
LIN {X 0,Y 345.423,Z 674.492,A -85,B 0,C 180,E1 -23284.362,E2 -23284.362} C_VEL
LIN {X 0,Y 349.591,Z 678.256,A -85,B 0,C 180,E1 -23286.915,E2 -23286.915} C_VEL
LIN {X 0,Y 353.554,Z 681.038,A -85,B 0,C 180,E1 -23289.527,E2 -23289.527} C_VEL
LIN {X 0,Y 356.864,Z 683.154,A -85,B 0,C 180,E1 -23291.923,E2 -23291.923} C_VEL
LIN {X 0,Y 359.59,Z 685.766,A -85,B 0,C 180,E1 -23294.296,E2 -23294.296} C_VEL
LIN {X 0,Y 362.23,Z 687.778,A -85,B 0,C 180,E1 -23296.847,E2 -23296.847} C_VEL
LIN {X 0,Y 364.22,Z 689.021,A -85,B 0,C 180,E1 -23299.171,E2 -23299.171} C_VEL
LIN {X 0,Y 366.12,Z 689.875,A -85,B 0,C 180,E1 -23301.815,E2 -23301.815} C_VEL
LIN {X 0,Y 367.472,Z 690.589,A -85,B 0,C 180,E1 -23304.513,E2 -23304.513} C_VEL
LIN {X 0,Y 368.22,Z 690.963,A -85,B 0,C 180,E1 -23306.718,E2 -23306.718} C_VEL
LIN {X 0,Y 368.543,Z 691.065,A -85,B 0,C 180,E1 -23308.907,E2 -23308.907} C_VEL
LIN {X 0,Y 368.543,Z 691.066,A -85,B 0,C 180,E1 -23311.093,E2 -23311.093} C_VEL
LIN {X 0,Y 368.22,Z 690.964,A -85,B 0,C 180,E1 -23313.282,E2 -23313.282} C_VEL
LIN {X 0,Y 367.329,Z 690.498,A -85,B 0,C 180,E1 -23315.794,E2 -23315.794} C_VEL
LIN {X 0,Y 365.963,Z 689.806,A -85,B 0,C 180,E1 -23318.461,E2 -23318.461} C_VEL
LIN {X 0,Y 363.979,Z 688.888,A -85,B 0,C 180,E1 -23321.133,E2 -23321.133} C_VEL
LIN {X 0,Y 361.451,Z 687.251,A -85,B 0,C 180,E1 -23323.928,E2 -23323.928} C_VEL
LIN {X 0,Y 358.798,Z 685.018,A -85,B 0,C 180,E1 -23326.445,E2 -23326.445} C_VEL
LIN {X 0,Y 356.074,Z 682.479,A -85,B 0,C 180,E1 -23328.668,E2 -23328.668} C_VEL
LIN {X 0,Y 352.463,Z 680.32,A -85,B 0,C 180,E1 -23331.232,E2 -23331.232} C_VEL
LIN {X 0,Y 348.237,Z 677.138,A -85,B 0,C 180,E1 -23333.951,E2 -23333.951} C_VEL
LIN {X 0,Y 344.907,Z 674.176,A -85,B 0,C 180,E1 -23335.921,E2 -23335.921} C_VEL
LIN {X 0,Y 340.644,Z 671.275,A -85,B 0,C 180,E1 -23338.244,E2 -23338.244} C_VEL
LIN {X 0,Y 335.705,Z 666.993,A -85,B 0,C 180,E1 -23340.794,E2 -23340.794} C_VEL
LIN {X 0,Y 329.528,Z 662.25,A -85,B 0,C 180,E1 -23343.72,E2 -23343.72} C_VEL
LIN {X 0,Y 324.548,Z 658.004,A -85,B 0,C 180,E1 -23345.975,E2 -23345.975} C_VEL
LIN {X 0,Y 318.457,Z 653.039,A -85,B 0,C 180,E1 -23348.595,E2 -23348.595} C_VEL
LIN {X 0,Y 313.694,Z 649.037,A -85,B 0,C 180,E1 -23350.562,E2 -23350.562} C_VEL
LIN {X 0,Y 307.868,Z 643.927,A -85,B 0,C 180,E1 -23352.867,E2 -23352.867} C_VEL
LIN {X 0,Y 300.692,Z 638.15,A -85,B 0,C 180,E1 -23355.418,E2 -23355.418} C_VEL
LIN {X 0,Y 293.745,Z 632.512,A -85,B 0,C 180,E1 -23357.671,E2 -23357.671} C_VEL
LIN {X 0,Y 286.268,Z 626.478,A -85,B 0,C 180,E1 -23359.918,E2 -23359.918} C_VEL
LIN {X 0,Y 272.122,Z 614.553,A -85,B 0,C 180,E1 -23364.188,E2 -23364.188} C_VEL
LIN {X 0,Y 264.27,Z 606.769,A -85,B 0,C 180,E1 -23367.021,E2 -23367.021} C_VEL
LIN {X 0,Y 256.612,Z 597.395,A -85,B 0,C 180,E1 -23370.299,E2 -23370.299} C_VEL
LIN {X 0,Y 249.052,Z 585.59,A -85,B 0,C 180,E1 -23374.301,E2 -23374.301} C_VEL
LIN {X 0,Y 244.673,Z 577.674,A -85,B 0,C 180,E1 -23377.129,E2 -23377.129} C_VEL
LIN {X 0,Y 240,Z 569.888,A -85,B 0,C 180,E1 -23380.655,E2 -23380.655} C_VEL
LIN {X 0,Y 237.85,Z 566.593,A -85,B 0,C 180,E1 -23382.534,E2 -23382.534} C_VEL
LIN {X 0,Y 235.248,Z 562.537,A -85,B 0,C 180,E1 -23385.179,E2 -23385.179} C_VEL
LIN {X 0,Y 232.983,Z 558.844,A -85,B 0,C 180,E1 -23388.031,E2 -23388.031} C_VEL
LIN {X 0,Y 230.717,Z 555.507,A -85,B 0,C 180,E1 -23391.846,E2 -23391.846} C_VEL
LIN {X 0,Y 230.275,Z 554.277,A -85,B 0,C 180,E1 -23392.988,E2 -23392.988} C_VEL
LIN {X 0,Y 228.837,Z 552.789,A -85,B 0,C 180,E1 -23400,E2 -23400} C_VEL
LIN {X 0,Y 230.379,Z 554.513,A -85,B 0,C 180,E1 -23406.868,E2 -23406.868} C_VEL
LIN {X 0,Y 232.207,Z 558.038,A -85,B 0,C 180,E1 -23410.463,E2 -23410.463} C_VEL
LIN {X 0,Y 233.352,Z 559.408,A -85,B 0,C 180,E1 -23412.061,E2 -23412.061} C_VEL
LIN {X 0,Y 236.089,Z 563.774,A -85,B 0,C 180,E1 -23415.306,E2 -23415.306} C_VEL
LIN {X 0,Y 239.367,Z 568.921,A -85,B 0,C 180,E1 -23418.399,E2 -23418.399} C_VEL
LIN {X 0,Y 242.938,Z 574.719,A -85,B 0,C 180,E1 -23421.222,E2 -23421.222} C_VEL
LIN {X 0,Y 245.755,Z 579.866,A -85,B 0,C 180,E1 -23423.211,E2 -23423.211} C_VEL
LIN {X 0,Y 249.31,Z 588.111,A -85,B 0,C 180,E1 -23425.571,E2 -23425.571} C_VEL
LIN {X 0,Y 252.741,Z 596.706,A -85,B 0,C 180,E1 -23427.654,E2 -23427.654} C_VEL
LIN {X 0,Y 253.261,Z 598.241,A -85,B 0,C 180,E1 -23427.966,E2 -23427.966} C_VEL
LIN {X 0,Y 245.803,Z 685.358,A -85,B 0,C 180,E1 -23430.029,E2 -23430.029} C_VEL
LIN {X 0,Y 243.826,Z 699.069,A -85,B 0,C 180,E1 -23430.459,E2 -23430.459} C_VEL
LIN {X 0,Y 241.293,Z 711.9,A -85,B 0,C 180,E1 -23430.975,E2 -23430.975} C_VEL
LIN {X 0,Y 238.28,Z 724.17,A -85,B 0,C 180,E1 -23431.609,E2 -23431.609} C_VEL
LIN {X 0,Y 235.022,Z 735.528,A -85,B 0,C 180,E1 -23432.354,E2 -23432.354} C_VEL
LIN {X 0,Y 231.134,Z 747.254,A -85,B 0,C 180,E1 -23433.29,E2 -23433.29} C_VEL
LIN {X 0,Y 226.716,Z 758.766,A -85,B 0,C 180,E1 -23434.378,E2 -23434.378} C_VEL
LIN {X 0,Y 221.785,Z 770.283,A -85,B 0,C 180,E1 -23435.709,E2 -23435.709} C_VEL
LIN {X 0,Y 216.391,Z 781.572,A -85,B 0,C 180,E1 -23437.279,E2 -23437.279} C_VEL
LIN {X 0,Y 210.568,Z 792.54,A -85,B 0,C 180,E1 -23439.106,E2 -23439.106} C_VEL
LIN {X 0,Y 205.092,Z 802.228,A -85,B 0,C 180,E1 -23441.073,E2 -23441.073} C_VEL
LIN {X 0,Y 198.729,Z 812.427,A -85,B 0,C 180,E1 -23443.534,E2 -23443.534} C_VEL
LIN {X 0,Y 192.834,Z 821.382,A -85,B 0,C 180,E1 -23446.175,E2 -23446.175} C_VEL
LIN {X 0,Y 187.305,Z 829.378,A -85,B 0,C 180,E1 -23449.021,E2 -23449.021} C_VEL
LIN {X 0,Y 182.44,Z 836.236,A -85,B 0,C 180,E1 -23451.951,E2 -23451.951} C_VEL
LIN {X 0,Y 177.943,Z 842.377,A -85,B 0,C 180,E1 -23455.063,E2 -23455.063} C_VEL
LIN {X 0,Y 172.791,Z 849.328,A -85,B 0,C 180,E1 -23459.442,E2 -23459.442} C_VEL
LIN {X 0,Y 168.661,Z 855.094,A -85,B 0,C 180,E1 -23464.054,E2 -23464.054} C_VEL
LIN {X 0,Y 167.589,Z 856.711,A -85,B 0,C 180,E1 -23465.546,E2 -23465.546} C_VEL
LIN {X 0,Y 165.749,Z 858.6,A -85,B 0,C 180,E1 -23467.364,E2 -23467.364} C_VEL
LIN {X 0,Y 161.229,Z 861.279,A -85,B 0,C 180,E1 -23470.315,E2 -23470.315} C_VEL
LIN {X 0,Y 157.702,Z 863.058,A -85,B 0,C 180,E1 -23472.809,E2 -23472.809} C_VEL
LIN {X 0,Y 155.798,Z 864.474,A -85,B 0,C 180,E1 -23475.195,E2 -23475.195} C_VEL
LIN {X 0,Y 155.677,Z 864.573,A -85,B 0,C 180,E1 -23475.551,E2 -23475.551} C_VEL
LIN {X 0,Y 154.919,Z 866.382,A -85,B 0,C 180,E1 -23479.545,E2 -23479.545} C_VEL
LIN {X 0,Y 154.637,Z 867.828,A -85,B 0,C 180,E1 -23484.785,E2 -23484.785} C_VEL
LIN {X 0,Y 154.774,Z 868.314,A -85,B 0,C 180,E1 -23490,E2 -23490} C_VEL
LIN {X 0,Y 154.637,Z 867.828,A -85,B 0,C 180,E1 -23495.215,E2 -23495.215} C_VEL
LIN {X 0,Y 154.917,Z 866.382,A -85,B 0,C 180,E1 -23500.455,E2 -23500.455} C_VEL
LIN {X 0,Y 156.041,Z 863.978,A -85,B 0,C 180,E1 -23505.678,E2 -23505.678} C_VEL
LIN {X 0,Y 158.537,Z 860.095,A -85,B 0,C 180,E1 -23511.418,E2 -23511.418} C_VEL
LIN {X 0,Y 161.282,Z 856.17,A -85,B 0,C 180,E1 -23515.833,E2 -23515.833} C_VEL
LIN {X 0,Y 165.42,Z 850.661,A -85,B 0,C 180,E1 -23520.652,E2 -23520.652} C_VEL
LIN {X 0,Y 169.817,Z 844.979,A -85,B 0,C 180,E1 -23524.611,E2 -23524.611} C_VEL
LIN {X 0,Y 175.185,Z 838.129,A -85,B 0,C 180,E1 -23528.448,E2 -23528.448} C_VEL
LIN {X 0,Y 180.285,Z 831.478,A -85,B 0,C 180,E1 -23531.505,E2 -23531.505} C_VEL
LIN {X 0,Y 185.753,Z 823.926,A -85,B 0,C 180,E1 -23534.422,E2 -23534.422} C_VEL
LIN {X 0,Y 191.721,Z 815.344,A -85,B 0,C 180,E1 -23537.149,E2 -23537.149} C_VEL
LIN {X 0,Y 197.069,Z 807.337,A -85,B 0,C 180,E1 -23539.272,E2 -23539.272} C_VEL
LIN {X 0,Y 204.285,Z 795.597,A -85,B 0,C 180,E1 -23541.803,E2 -23541.803} C_VEL
LIN {X 0,Y 209.685,Z 785.931,A -85,B 0,C 180,E1 -23543.551,E2 -23543.551} C_VEL
LIN {X 0,Y 215.784,Z 773.983,A -85,B 0,C 180,E1 -23545.322,E2 -23545.322} C_VEL
LIN {X 0,Y 220.861,Z 763.053,A -85,B 0,C 180,E1 -23546.645,E2 -23546.645} C_VEL
LIN {X 0,Y 225.916,Z 750.671,A -85,B 0,C 180,E1 -23547.898,E2 -23547.898} C_VEL
LIN {X 0,Y 230.268,Z 738.393,A -85,B 0,C 180,E1 -23548.923,E2 -23548.923} C_VEL
LIN {X 0,Y 234.312,Z 725.195,A -85,B 0,C 180,E1 -23549.79,E2 -23549.79} C_VEL
LIN {X 0,Y 237.562,Z 712.458,A -85,B 0,C 180,E1 -23550.451,E2 -23550.451} C_VEL
LIN {X 0,Y 240.135,Z 699.858,A -85,B 0,C 180,E1 -23550.966,E2 -23550.966} C_VEL
LIN {X 0,Y 242.06,Z 687.072,A -85,B 0,C 180,E1 -23551.382,E2 -23551.382} C_VEL
LIN {X 0,Y 245.018,Z 655.648,A -85,B 0,C 180,E1 -23552.142,E2 -23552.142} C_VEL
LIN {X 0,Y 249.737,Z 601.259,A -85,B 0,C 180,E1 -23553.394,E2 -23553.394} C_VEL
LIN {X 0,Y 245.402,Z 590.032,A -85,B 0,C 180,E1 -23556.252,E2 -23556.252} C_VEL
LIN {X 0,Y 242.476,Z 583.518,A -85,B 0,C 180,E1 -23558.362,E2 -23558.362} C_VEL
LIN {X 0,Y 238.592,Z 576.782,A -85,B 0,C 180,E1 -23561.428,E2 -23561.428} C_VEL
LIN {X 0,Y 236.318,Z 573.14,A -85,B 0,C 180,E1 -23563.496,E2 -23563.496} C_VEL
LIN {X 0,Y 233.98,Z 569.284,A -85,B 0,C 180,E1 -23565.987,E2 -23565.987} C_VEL
LIN {X 0,Y 231.789,Z 565.676,A -85,B 0,C 180,E1 -23568.855,E2 -23568.855} C_VEL
LIN {X 0,Y 229.534,Z 562.019,A -85,B 0,C 180,E1 -23572.965,E2 -23572.965} C_VEL
LIN {X 0,Y 229.319,Z 561.288,A -85,B 0,C 180,E1 -23573.593,E2 -23573.593} C_VEL
LIN {X 0,Y 227.973,Z 559.823,A -85,B 0,C 180,E1 -23580,E2 -23580} C_VEL
LIN {X 0,Y 229.355,Z 561.397,A -85,B 0,C 180,E1 -23586.929,E2 -23586.929} C_VEL
LIN {X 0,Y 231.077,Z 564.898,A -85,B 0,C 180,E1 -23590.514,E2 -23590.514} C_VEL
LIN {X 0,Y 232.174,Z 566.332,A -85,B 0,C 180,E1 -23592.122,E2 -23592.122} C_VEL
LIN {X 0,Y 234.836,Z 570.779,A -85,B 0,C 180,E1 -23595.402,E2 -23595.402} C_VEL
LIN {X 0,Y 237.724,Z 575.358,A -85,B 0,C 180,E1 -23598.227,E2 -23598.227} C_VEL
LIN {X 0,Y 241.107,Z 581.111,A -85,B 0,C 180,E1 -23601.031,E2 -23601.031} C_VEL
LIN {X 0,Y 245.15,Z 588.446,A -85,B 0,C 180,E1 -23603.918,E2 -23603.918} C_VEL
LIN {X 0,Y 253.735,Z 602.831,A -85,B 0,C 180,E1 -23608.847,E2 -23608.847} C_VEL
LIN {X 0,Y 260.309,Z 611.188,A -85,B 0,C 180,E1 -23611.828,E2 -23611.828} C_VEL
LIN {X 0,Y 267.983,Z 619.332,A -85,B 0,C 180,E1 -23614.778,E2 -23614.778} C_VEL
LIN {X 0,Y 284.607,Z 633.506,A -85,B 0,C 180,E1 -23619.943,E2 -23619.943} C_VEL
LIN {X 0,Y 293.034,Z 640.221,A -85,B 0,C 180,E1 -23622.457,E2 -23622.457} C_VEL
LIN {X 0,Y 298.994,Z 645.02,A -85,B 0,C 180,E1 -23624.388,E2 -23624.388} C_VEL
LIN {X 0,Y 305.774,Z 650.366,A -85,B 0,C 180,E1 -23626.739,E2 -23626.739} C_VEL
LIN {X 0,Y 312.403,Z 656.122,A -85,B 0,C 180,E1 -23629.323,E2 -23629.323} C_VEL
LIN {X 0,Y 317.603,Z 660.471,A -85,B 0,C 180,E1 -23631.465,E2 -23631.465} C_VEL
LIN {X 0,Y 323.355,Z 665.022,A -85,B 0,C 180,E1 -23633.926,E2 -23633.926} C_VEL
LIN {X 0,Y 329.493,Z 670.211,A -85,B 0,C 180,E1 -23636.702,E2 -23636.702} C_VEL
LIN {X 0,Y 334.483,Z 673.985,A -85,B 0,C 180,E1 -23639.076,E2 -23639.076} C_VEL
LIN {X 0,Y 339.523,Z 678.333,A -85,B 0,C 180,E1 -23641.663,E2 -23641.663} C_VEL
LIN {X 0,Y 344.086,Z 681.365,A -85,B 0,C 180,E1 -23644.134,E2 -23644.134} C_VEL
LIN {X 0,Y 348.332,Z 685.116,A -85,B 0,C 180,E1 -23646.696,E2 -23646.696} C_VEL
LIN {X 0,Y 352.628,Z 688.11,A -85,B 0,C 180,E1 -23649.507,E2 -23649.507} C_VEL
LIN {X 0,Y 355.792,Z 690.139,A -85,B 0,C 180,E1 -23651.794,E2 -23651.794} C_VEL
LIN {X 0,Y 358.658,Z 692.801,A -85,B 0,C 180,E1 -23654.255,E2 -23654.255} C_VEL
LIN {X 0,Y 361.324,Z 694.835,A -85,B 0,C 180,E1 -23656.814,E2 -23656.814} C_VEL
LIN {X 0,Y 363.515,Z 696.14,A -85,B 0,C 180,E1 -23659.374,E2 -23659.374} C_VEL
LIN {X 0,Y 365.24,Z 696.919,A -85,B 0,C 180,E1 -23661.795,E2 -23661.795} C_VEL
LIN {X 0,Y 366.599,Z 697.615,A -85,B 0,C 180,E1 -23664.5,E2 -23664.5} C_VEL
LIN {X 0,Y 367.353,Z 698.009,A -85,B 0,C 180,E1 -23666.71,E2 -23666.71} C_VEL
LIN {X 0,Y 367.677,Z 698.112,A -85,B 0,C 180,E1 -23668.905,E2 -23668.905} C_VEL
LIN {X 0,Y 367.677,Z 698.112,A -85,B 0,C 180,E1 -23671.095,E2 -23671.095} C_VEL
LIN {X 0,Y 367.353,Z 698.01,A -85,B 0,C 180,E1 -23673.29,E2 -23673.29} C_VEL
LIN {X 0,Y 366.455,Z 697.529,A -85,B 0,C 180,E1 -23675.808,E2 -23675.808} C_VEL
LIN {X 0,Y 365.081,Z 696.85,A -85,B 0,C 180,E1 -23678.482,E2 -23678.482} C_VEL
LIN {X 0,Y 363.083,Z 695.928,A -85,B 0,C 180,E1 -23681.161,E2 -23681.161} C_VEL
LIN {X 0,Y 360.57,Z 694.298,A -85,B 0,C 180,E1 -23683.929,E2 -23683.929} C_VEL
LIN {X 0,Y 357.829,Z 692.053,A -85,B 0,C 180,E1 -23686.516,E2 -23686.516} C_VEL
LIN {X 0,Y 354.904,Z 689.405,A -85,B 0,C 180,E1 -23688.873,E2 -23688.873} C_VEL
LIN {X 0,Y 351.219,Z 687.196,A -85,B 0,C 180,E1 -23691.449,E2 -23691.449} C_VEL
LIN {X 0,Y 347.068,Z 684.088,A -85,B 0,C 180,E1 -23694.098,E2 -23694.098} C_VEL
LIN {X 0,Y 343.422,Z 680.924,A -85,B 0,C 180,E1 -23696.239,E2 -23696.239} C_VEL
LIN {X 0,Y 339.305,Z 678.141,A -85,B 0,C 180,E1 -23698.45,E2 -23698.45} C_VEL
LIN {X 0,Y 334.479,Z 674.007,A -85,B 0,C 180,E1 -23700.924,E2 -23700.924} C_VEL
LIN {X 0,Y 328.164,Z 669.162,A -85,B 0,C 180,E1 -23703.906,E2 -23703.906} C_VEL
LIN {X 0,Y 323.164,Z 664.898,A -85,B 0,C 180,E1 -23706.157,E2 -23706.157} C_VEL
LIN {X 0,Y 317.355,Z 660.231,A -85,B 0,C 180,E1 -23708.639,E2 -23708.639} C_VEL
LIN {X 0,Y 311.5,Z 655.332,A -85,B 0,C 180,E1 -23711.043,E2 -23711.043} C_VEL
LIN {X 0,Y 304.893,Z 649.67,A -85,B 0,C 180,E1 -23713.571,E2 -23713.571} C_VEL
LIN {X 0,Y 298.819,Z 644.911,A -85,B 0,C 180,E1 -23715.668,E2 -23715.668} C_VEL
LIN {X 0,Y 293.841,Z 640.82,A -85,B 0,C 180,E1 -23717.292,E2 -23717.292} C_VEL
LIN {X 0,Y 287.211,Z 635.404,A -85,B 0,C 180,E1 -23719.315,E2 -23719.315} C_VEL
LIN {X 0,Y 279.135,Z 629.109,A -85,B 0,C 180,E1 -23721.627,E2 -23721.627} C_VEL
LIN {X 0,Y 269.364,Z 620.551,A -85,B 0,C 180,E1 -23724.742,E2 -23724.742} C_VEL
LIN {X 0,Y 261.958,Z 613.14,A -85,B 0,C 180,E1 -23727.493,E2 -23727.493} C_VEL
LIN {X 0,Y 254.301,Z 603.615,A -85,B 0,C 180,E1 -23730.875,E2 -23730.875} C_VEL
LIN {X 0,Y 246.744,Z 591.48,A -85,B 0,C 180,E1 -23735.046,E2 -23735.046} C_VEL
LIN {X 0,Y 242.575,Z 583.686,A -85,B 0,C 180,E1 -23737.875,E2 -23737.875} C_VEL
LIN {X 0,Y 238.259,Z 576.22,A -85,B 0,C 180,E1 -23741.302,E2 -23741.302} C_VEL
LIN {X 0,Y 236.174,Z 572.939,A -85,B 0,C 180,E1 -23743.218,E2 -23743.218} C_VEL
LIN {X 0,Y 233.726,Z 568.963,A -85,B 0,C 180,E1 -23745.859,E2 -23745.859} C_VEL
LIN {X 0,Y 231.655,Z 565.532,A -85,B 0,C 180,E1 -23748.627,E2 -23748.627} C_VEL
LIN {X 0,Y 229.543,Z 562.048,A -85,B 0,C 180,E1 -23752.524,E2 -23752.524} C_VEL
LIN {X 0,Y 229.23,Z 561.193,A -85,B 0,C 180,E1 -23753.398,E2 -23753.398} C_VEL
LIN {X 0,Y 227.971,Z 559.84,A -85,B 0,C 180,E1 -23760,E2 -23760} C_VEL
LIN {X 0,Y 229.375,Z 561.453,A -85,B 0,C 180,E1 -23766.571,E2 -23766.571} C_VEL
LIN {X 0,Y 231.061,Z 564.879,A -85,B 0,C 180,E1 -23770.073,E2 -23770.073} C_VEL
LIN {X 0,Y 232.16,Z 566.268,A -85,B 0,C 180,E1 -23771.68,E2 -23771.68} C_VEL
LIN {X 0,Y 234.801,Z 570.638,A -85,B 0,C 180,E1 -23774.939,E2 -23774.939} C_VEL
LIN {X 0,Y 237.798,Z 575.524,A -85,B 0,C 180,E1 -23777.882,E2 -23777.882} C_VEL
LIN {X 0,Y 240.882,Z 580.684,A -85,B 0,C 180,E1 -23780.439,E2 -23780.439} C_VEL
LIN {X 0,Y 243.664,Z 585.989,A -85,B 0,C 180,E1 -23782.51,E2 -23782.51} C_VEL
LIN {X 0,Y 247.251,Z 594.683,A -85,B 0,C 180,E1 -23785.007,E2 -23785.007} C_VEL
LIN {X 0,Y 249.717,Z 601.213,A -85,B 0,C 180,E1 -23786.594,E2 -23786.594} C_VEL
LIN {X 0,Y 242.378,Z 684.579,A -85,B 0,C 180,E1 -23788.551,E2 -23788.551} C_VEL
LIN {X 0,Y 240.468,Z 697.859,A -85,B 0,C 180,E1 -23788.962,E2 -23788.962} C_VEL
LIN {X 0,Y 237.893,Z 710.925,A -85,B 0,C 180,E1 -23789.475,E2 -23789.475} C_VEL
LIN {X 0,Y 234.961,Z 722.725,A -85,B 0,C 180,E1 -23790.056,E2 -23790.056} C_VEL
LIN {X 0,Y 231.283,Z 735.318,A -85,B 0,C 180,E1 -23790.861,E2 -23790.861} C_VEL
LIN {X 0,Y 226.901,Z 748.096,A -85,B 0,C 180,E1 -23791.881,E2 -23791.881} C_VEL
LIN {X 0,Y 222.12,Z 760.054,A -85,B 0,C 180,E1 -23793.023,E2 -23793.023} C_VEL
LIN {X 0,Y 217.058,Z 771.376,A -85,B 0,C 180,E1 -23794.348,E2 -23794.348} C_VEL
LIN {X 0,Y 211.522,Z 782.503,A -85,B 0,C 180,E1 -23795.918,E2 -23795.918} C_VEL
LIN {X 0,Y 205.543,Z 793.335,A -85,B 0,C 180,E1 -23797.751,E2 -23797.751} C_VEL
LIN {X 0,Y 199.344,Z 803.791,A -85,B 0,C 180,E1 -23799.933,E2 -23799.933} C_VEL
LIN {X 0,Y 193.836,Z 812.215,A -85,B 0,C 180,E1 -23801.99,E2 -23801.99} C_VEL
LIN {X 0,Y 187.707,Z 821.169,A -85,B 0,C 180,E1 -23804.654,E2 -23804.654} C_VEL
LIN {X 0,Y 181.809,Z 829.288,A -85,B 0,C 180,E1 -23807.576,E2 -23807.576} C_VEL
LIN {X 0,Y 176.83,Z 836.024,A -85,B 0,C 180,E1 -23810.513,E2 -23810.513} C_VEL
LIN {X 0,Y 172.075,Z 842.164,A -85,B 0,C 180,E1 -23813.686,E2 -23813.686} C_VEL
LIN {X 0,Y 166.618,Z 849.115,A -85,B 0,C 180,E1 -23818.181,E2 -23818.181} C_VEL
LIN {X 0,Y 162.204,Z 854.881,A -85,B 0,C 180,E1 -23822.939,E2 -23822.939} C_VEL
LIN {X 0,Y 159.613,Z 858.504,A -85,B 0,C 180,E1 -23826.655,E2 -23826.655} C_VEL
LIN {X 0,Y 157.013,Z 862.37,A -85,B 0,C 180,E1 -23831.741,E2 -23831.741} C_VEL
LIN {X 0,Y 155.677,Z 864.573,A -85,B 0,C 180,E1 -23835.551,E2 -23835.551} C_VEL
LIN {X 0,Y 154.514,Z 865.571,A -85,B 0,C 180,E1 -23837.66,E2 -23837.66} C_VEL
LIN {X 0,Y 152.59,Z 866.455,A -85,B 0,C 180,E1 -23839.737,E2 -23839.737} C_VEL
LIN {X 0,Y 148.59,Z 867.508,A -85,B 0,C 180,E1 -23844.009,E2 -23844.009} C_VEL
LIN {X 0,Y 147.593,Z 867.805,A -85,B 0,C 180,E1 -23846.276,E2 -23846.276} C_VEL
LIN {X 0,Y 147.552,Z 867.865,A -85,B 0,C 180,E1 -23847.046,E2 -23847.046} C_VEL
LIN {X 0,Y 147.677,Z 868.104,A -85,B 0,C 180,E1 -23850,E2 -23850} C_VEL
LIN {X 0,Y 147.54,Z 867.617,A -85,B 0,C 180,E1 -23855.467,E2 -23855.467} C_VEL
LIN {X 0,Y 147.893,Z 866.171,A -85,B 0,C 180,E1 -23860.957,E2 -23860.957} C_VEL
LIN {X 0,Y 149.138,Z 863.766,A -85,B 0,C 180,E1 -23866.424,E2 -23866.424} C_VEL
LIN {X 0,Y 151.653,Z 860.167,A -85,B 0,C 180,E1 -23872.05,E2 -23872.05} C_VEL
LIN {X 0,Y 154.801,Z 855.957,A -85,B 0,C 180,E1 -23877,E2 -23877} C_VEL
LIN {X 0,Y 159.228,Z 850.447,A -85,B 0,C 180,E1 -23881.981,E2 -23881.981} C_VEL
LIN {X 0,Y 163.262,Z 845.585,A -85,B 0,C 180,E1 -23885.528,E2 -23885.528} C_VEL
LIN {X 0,Y 169.594,Z 837.916,A -85,B 0,C 180,E1 -23889.964,E2 -23889.964} C_VEL
LIN {X 0,Y 174.926,Z 831.264,A -85,B 0,C 180,E1 -23893.078,E2 -23893.078} C_VEL
LIN {X 0,Y 180.676,Z 823.713,A -85,B 0,C 180,E1 -23896.022,E2 -23896.022} C_VEL
LIN {X 0,Y 186.909,Z 815.132,A -85,B 0,C 180,E1 -23898.765,E2 -23898.765} C_VEL
LIN {X 0,Y 193.623,Z 805.351,A -85,B 0,C 180,E1 -23901.295,E2 -23901.295} C_VEL
LIN {X 0,Y 199.939,Z 795.368,A -85,B 0,C 180,E1 -23903.422,E2 -23903.422} C_VEL
LIN {X 0,Y 205.507,Z 785.719,A -85,B 0,C 180,E1 -23905.159,E2 -23905.159} C_VEL
LIN {X 0,Y 211.804,Z 773.772,A -85,B 0,C 180,E1 -23906.91,E2 -23906.91} C_VEL
LIN {X 0,Y 217.009,Z 762.842,A -85,B 0,C 180,E1 -23908.223,E2 -23908.223} C_VEL
LIN {X 0,Y 222.237,Z 750.4,A -85,B 0,C 180,E1 -23909.458,E2 -23909.458} C_VEL
LIN {X 0,Y 226.678,Z 738.183,A -85,B 0,C 180,E1 -23910.463,E2 -23910.463} C_VEL
LIN {X 0,Y 230.822,Z 724.985,A -85,B 0,C 180,E1 -23911.313,E2 -23911.313} C_VEL
LIN {X 0,Y 234.146,Z 712.248,A -85,B 0,C 180,E1 -23911.96,E2 -23911.96} C_VEL
LIN {X 0,Y 236.762,Z 699.648,A -85,B 0,C 180,E1 -23912.472,E2 -23912.472} C_VEL
LIN {X 0,Y 238.788,Z 686.285,A -85,B 0,C 180,E1 -23912.903,E2 -23912.903} C_VEL
LIN {X 0,Y 242.401,Z 648.717,A -85,B 0,C 180,E1 -23913.774,E2 -23913.774} C_VEL
LIN {X 0,Y 246.294,Z 604.401,A -85,B 0,C 180,E1 -23914.815,E2 -23914.815} C_VEL
LIN {X 0,Y 242.698,Z 594.816,A -85,B 0,C 180,E1 -23917.372,E2 -23917.372} C_VEL
LIN {X 0,Y 240.356,Z 589.393,A -85,B 0,C 180,E1 -23919.175,E2 -23919.175} C_VEL
LIN {X 0,Y 236.647,Z 582.78,A -85,B 0,C 180,E1 -23922.277,E2 -23922.277} C_VEL
LIN {X 0,Y 234.512,Z 579.229,A -85,B 0,C 180,E1 -23924.352,E2 -23924.352} C_VEL
LIN {X 0,Y 232.561,Z 575.88,A -85,B 0,C 180,E1 -23926.566,E2 -23926.566} C_VEL
LIN {X 0,Y 230.479,Z 572.346,A -85,B 0,C 180,E1 -23929.458,E2 -23929.458} C_VEL
LIN {X 0,Y 228.454,Z 568.736,A -85,B 0,C 180,E1 -23933.474,E2 -23933.474} C_VEL
LIN {X 0,Y 228.299,Z 568.26,A -85,B 0,C 180,E1 -23933.943,E2 -23933.943} C_VEL
LIN {X 0,Y 227.108,Z 566.87,A -85,B 0,C 180,E1 -23940,E2 -23940} C_VEL
LIN {X 0,Y 228.356,Z 568.352,A -85,B 0,C 180,E1 -23946.627,E2 -23946.627} C_VEL
LIN {X 0,Y 230.075,Z 571.906,A -85,B 0,C 180,E1 -23950.338,E2 -23950.338} C_VEL
LIN {X 0,Y 230.994,Z 573.182,A -85,B 0,C 180,E1 -23951.739,E2 -23951.739} C_VEL
LIN {X 0,Y 233.474,Z 577.488,A -85,B 0,C 180,E1 -23954.936,E2 -23954.936} C_VEL
LIN {X 0,Y 236.34,Z 582.187,A -85,B 0,C 180,E1 -23957.849,E2 -23957.849} C_VEL
LIN {X 0,Y 240.255,Z 589.241,A -85,B 0,C 180,E1 -23961.166,E2 -23961.166} C_VEL
LIN {X 0,Y 243.944,Z 596.278,A -85,B 0,C 180,E1 -23963.835,E2 -23963.835} C_VEL
LIN {X 0,Y 251.192,Z 608.638,A -85,B 0,C 180,E1 -23968.116,E2 -23968.116} C_VEL
LIN {X 0,Y 257.829,Z 617.336,A -85,B 0,C 180,E1 -23971.248,E2 -23971.248} C_VEL
LIN {X 0,Y 265.619,Z 625.697,A -85,B 0,C 180,E1 -23974.333,E2 -23974.333} C_VEL
LIN {X 0,Y 282.288,Z 640.009,A -85,B 0,C 180,E1 -23979.613,E2 -23979.613} C_VEL
LIN {X 0,Y 290.555,Z 646.56,A -85,B 0,C 180,E1 -23982.044,E2 -23982.044} C_VEL
LIN {X 0,Y 296.017,Z 650.874,A -85,B 0,C 180,E1 -23983.766,E2 -23983.766} C_VEL
LIN {X 0,Y 302.12,Z 655.672,A -85,B 0,C 180,E1 -23985.829,E2 -23985.829} C_VEL
LIN {X 0,Y 307.737,Z 660.472,A -85,B 0,C 180,E1 -23987.909,E2 -23987.909} C_VEL
LIN {X 0,Y 314.234,Z 665.706,A -85,B 0,C 180,E1 -23990.479,E2 -23990.479} C_VEL
LIN {X 0,Y 320.057,Z 670.547,A -85,B 0,C 180,E1 -23992.929,E2 -23992.929} C_VEL
LIN {X 0,Y 324.168,Z 673.778,A -85,B 0,C 180,E1 -23994.711,E2 -23994.711} C_VEL
LIN {X 0,Y 329.514,Z 678.135,A -85,B 0,C 180,E1 -23997.155,E2 -23997.155} C_VEL
LIN {X 0,Y 333.176,Z 680.924,A -85,B 0,C 180,E1 -23998.906,E2 -23998.906} C_VEL
LIN {X 0,Y 337.908,Z 684.962,A -85,B 0,C 180,E1 -24001.311,E2 -24001.311} C_VEL
LIN {X 0,Y 342.501,Z 688.077,A -85,B 0,C 180,E1 -24003.762,E2 -24003.762} C_VEL
LIN {X 0,Y 347.076,Z 691.976,A -85,B 0,C 180,E1 -24006.476,E2 -24006.476} C_VEL
LIN {X 0,Y 351.38,Z 694.964,A -85,B 0,C 180,E1 -24009.253,E2 -24009.253} C_VEL
LIN {X 0,Y 354.752,Z 697.134,A -85,B 0,C 180,E1 -24011.69,E2 -24011.69} C_VEL
LIN {X 0,Y 357.52,Z 699.701,A -85,B 0,C 180,E1 -24014.026,E2 -24014.026} C_VEL
LIN {X 0,Y 360.25,Z 701.774,A -85,B 0,C 180,E1 -24016.608,E2 -24016.608} C_VEL
LIN {X 0,Y 362.184,Z 702.99,A -85,B 0,C 180,E1 -24018.811,E2 -24018.811} C_VEL
LIN {X 0,Y 364.199,Z 703.886,A -85,B 0,C 180,E1 -24021.496,E2 -24021.496} C_VEL
LIN {X 0,Y 365.553,Z 704.555,A -85,B 0,C 180,E1 -24024.115,E2 -24024.115} C_VEL
LIN {X 0,Y 366.486,Z 705.055,A -85,B 0,C 180,E1 -24026.702,E2 -24026.702} C_VEL
LIN {X 0,Y 366.811,Z 705.158,A -85,B 0,C 180,E1 -24028.902,E2 -24028.902} C_VEL
LIN {X 0,Y 366.811,Z 705.158,A -85,B 0,C 180,E1 -24031.098,E2 -24031.098} C_VEL
LIN {X 0,Y 366.292,Z 704.972,A -85,B 0,C 180,E1 -24033.881,E2 -24033.881} C_VEL
LIN {X 0,Y 365.396,Z 704.46,A -85,B 0,C 180,E1 -24036.256,E2 -24036.256} C_VEL
LIN {X 0,Y 363.918,Z 703.73,A -85,B 0,C 180,E1 -24038.887,E2 -24038.887} C_VEL
LIN {X 0,Y 361.986,Z 702.83,A -85,B 0,C 180,E1 -24041.46,E2 -24041.46} C_VEL
LIN {X 0,Y 359.455,Z 701.22,A -85,B 0,C 180,E1 -24044.155,E2 -24044.155} C_VEL
LIN {X 0,Y 356.619,Z 698.874,A -85,B 0,C 180,E1 -24046.773,E2 -24046.773} C_VEL
LIN {X 0,Y 353.736,Z 696.331,A -85,B 0,C 180,E1 -24049.081,E2 -24049.081} C_VEL
LIN {X 0,Y 349.99,Z 694.068,A -85,B 0,C 180,E1 -24051.66,E2 -24051.66} C_VEL
LIN {X 0,Y 345.77,Z 690.94,A -85,B 0,C 180,E1 -24054.317,E2 -24054.317} C_VEL
LIN {X 0,Y 342.107,Z 687.797,A -85,B 0,C 180,E1 -24056.466,E2 -24056.466} C_VEL
LIN {X 0,Y 337.91,Z 684.954,A -85,B 0,C 180,E1 -24058.688,E2 -24058.688} C_VEL
LIN {X 0,Y 332.963,Z 680.726,A -85,B 0,C 180,E1 -24061.199,E2 -24061.199} C_VEL
LIN {X 0,Y 326.882,Z 676.113,A -85,B 0,C 180,E1 -24064.057,E2 -24064.057} C_VEL
LIN {X 0,Y 321.208,Z 671.384,A -85,B 0,C 180,E1 -24066.585,E2 -24066.585} C_VEL
LIN {X 0,Y 314.857,Z 666.27,A -85,B 0,C 180,E1 -24069.265,E2 -24069.265} C_VEL
LIN {X 0,Y 309.109,Z 661.519,A -85,B 0,C 180,E1 -24071.57,E2 -24071.57} C_VEL
LIN {X 0,Y 303.795,Z 656.988,A -85,B 0,C 180,E1 -24073.578,E2 -24073.578} C_VEL
LIN {X 0,Y 297.605,Z 652.216,A -85,B 0,C 180,E1 -24075.702,E2 -24075.702} C_VEL
LIN {X 0,Y 291.961,Z 647.57,A -85,B 0,C 180,E1 -24077.526,E2 -24077.526} C_VEL
LIN {X 0,Y 285.124,Z 642.143,A -85,B 0,C 180,E1 -24079.574,E2 -24079.574} C_VEL
LIN {X 0,Y 275.646,Z 634.557,A -85,B 0,C 180,E1 -24082.33,E2 -24082.33} C_VEL
LIN {X 0,Y 267.665,Z 627.607,A -85,B 0,C 180,E1 -24084.938,E2 -24084.938} C_VEL
LIN {X 0,Y 259.357,Z 619.135,A -85,B 0,C 180,E1 -24088.103,E2 -24088.103} C_VEL
LIN {X 0,Y 251.842,Z 609.567,A -85,B 0,C 180,E1 -24091.551,E2 -24091.551} C_VEL
LIN {X 0,Y 244.681,Z 597.755,A -85,B 0,C 180,E1 -24095.67,E2 -24095.67} C_VEL
LIN {X 0,Y 240.652,Z 589.912,A -85,B 0,C 180,E1 -24098.534,E2 -24098.534} C_VEL
LIN {X 0,Y 236.479,Z 582.451,A -85,B 0,C 180,E1 -24102.02,E2 -24102.02} C_VEL
LIN {X 0,Y 234.532,Z 579.325,A -85,B 0,C 180,E1 -24103.908,E2 -24103.908} C_VEL
LIN {X 0,Y 232.495,Z 575.794,A -85,B 0,C 180,E1 -24106.229,E2 -24106.229} C_VEL
LIN {X 0,Y 230.494,Z 572.394,A -85,B 0,C 180,E1 -24109.014,E2 -24109.014} C_VEL
LIN {X 0,Y 228.423,Z 568.624,A -85,B 0,C 180,E1 -24113.153,E2 -24113.153} C_VEL
LIN {X 0,Y 228.191,Z 568.151,A -85,B 0,C 180,E1 -24113.812,E2 -24113.812} C_VEL
LIN {X 0,Y 227.106,Z 566.892,A -85,B 0,C 180,E1 -24120,E2 -24120} C_VEL
LIN {X 0,Y 228.391,Z 568.473,A -85,B 0,C 180,E1 -24126.32,E2 -24126.32} C_VEL
LIN {X 0,Y 230.05,Z 571.882,A -85,B 0,C 180,E1 -24129.884,E2 -24129.884} C_VEL
LIN {X 0,Y 230.982,Z 573.099,A -85,B 0,C 180,E1 -24131.296,E2 -24131.296} C_VEL
LIN {X 0,Y 233.425,Z 577.332,A -85,B 0,C 180,E1 -24134.455,E2 -24134.455} C_VEL
LIN {X 0,Y 236.201,Z 582.024,A -85,B 0,C 180,E1 -24137.31,E2 -24137.31} C_VEL
LIN {X 0,Y 239.316,Z 587.515,A -85,B 0,C 180,E1 -24140.009,E2 -24140.009} C_VEL
LIN {X 0,Y 241.602,Z 592.107,A -85,B 0,C 180,E1 -24141.793,E2 -24141.793} C_VEL
LIN {X 0,Y 245.101,Z 601.055,A -85,B 0,C 180,E1 -24144.361,E2 -24144.361} C_VEL
LIN {X 0,Y 246.32,Z 604.356,A -85,B 0,C 180,E1 -24145.195,E2 -24145.195} C_VEL
LIN {X 0,Y 238.97,Z 685.16,A -85,B 0,C 180,E1 -24147.078,E2 -24147.078} C_VEL
LIN {X 0,Y 236.94,Z 698.649,A -85,B 0,C 180,E1 -24147.496,E2 -24147.496} C_VEL
LIN {X 0,Y 234.302,Z 711.481,A -85,B 0,C 180,E1 -24147.997,E2 -24147.997} C_VEL
LIN {X 0,Y 231.142,Z 723.75,A -85,B 0,C 180,E1 -24148.605,E2 -24148.605} C_VEL
LIN {X 0,Y 227.375,Z 736.133,A -85,B 0,C 180,E1 -24149.397,E2 -24149.397} C_VEL
LIN {X 0,Y 223.203,Z 747.884,A -85,B 0,C 180,E1 -24150.32,E2 -24150.32} C_VEL
LIN {X 0,Y 218.316,Z 759.843,A -85,B 0,C 180,E1 -24151.453,E2 -24151.453} C_VEL
LIN {X 0,Y 213.091,Z 771.164,A -85,B 0,C 180,E1 -24152.754,E2 -24152.754} C_VEL
LIN {X 0,Y 207.419,Z 782.292,A -85,B 0,C 180,E1 -24154.322,E2 -24154.322} C_VEL
LIN {X 0,Y 201.227,Z 793.123,A -85,B 0,C 180,E1 -24156.134,E2 -24156.134} C_VEL
LIN {X 0,Y 195.958,Z 801.804,A -85,B 0,C 180,E1 -24157.907,E2 -24157.907} C_VEL
LIN {X 0,Y 189.102,Z 812.002,A -85,B 0,C 180,E1 -24160.371,E2 -24160.371} C_VEL
LIN {X 0,Y 182.709,Z 820.956,A -85,B 0,C 180,E1 -24163.044,E2 -24163.044} C_VEL
LIN {X 0,Y 176.312,Z 829.379,A -85,B 0,C 180,E1 -24166.121,E2 -24166.121} C_VEL
LIN {X 0,Y 171.327,Z 835.811,A -85,B 0,C 180,E1 -24168.98,E2 -24168.98} C_VEL
LIN {X 0,Y 166.308,Z 841.95,A -85,B 0,C 180,E1 -24172.212,E2 -24172.212} C_VEL
LIN {X 0,Y 160.526,Z 848.901,A -85,B 0,C 180,E1 -24176.821,E2 -24176.821} C_VEL
LIN {X 0,Y 155.797,Z 854.667,A -85,B 0,C 180,E1 -24181.729,E2 -24181.729} C_VEL
LIN {X 0,Y 153.011,Z 858.291,A -85,B 0,C 180,E1 -24185.583,E2 -24185.583} C_VEL
LIN {X 0,Y 150.199,Z 862.157,A -85,B 0,C 180,E1 -24190.881,E2 -24190.881} C_VEL
LIN {X 0,Y 148.359,Z 865.024,A -85,B 0,C 180,E1 -24196.299,E2 -24196.299} C_VEL
LIN {X 0,Y 147.895,Z 866.171,A -85,B 0,C 180,E1 -24199.043,E2 -24199.043} C_VEL
LIN {X 0,Y 147.54,Z 867.617,A -85,B 0,C 180,E1 -24204.533,E2 -24204.533} C_VEL
LIN {X 0,Y 147.552,Z 867.865,A -85,B 0,C 180,E1 -24207.046,E2 -24207.046} C_VEL
LIN {X 0,Y 146.955,Z 868.059,A -85,B 0,C 180,E1 -24209.321,E2 -24209.321} C_VEL
LIN {X 0,Y 145.358,Z 867.957,A -85,B 0,C 180,E1 -24211.564,E2 -24211.564} C_VEL
LIN {X 0,Y 141.576,Z 867.336,A -85,B 0,C 180,E1 -24216.136,E2 -24216.136} C_VEL
LIN {X 0,Y 140.607,Z 866.745,A -85,B 0,C 180,E1 -24218.542,E2 -24218.542} C_VEL
LIN {X 0,Y 140.58,Z 866.527,A -85,B 0,C 180,E1 -24219.356,E2 -24219.356} C_VEL
LIN {X 0,Y 141.385,Z 864.812,A -85,B 0,C 180,E1 -24224.391,E2 -24224.391} C_VEL
LIN {X 0,Y 143.42,Z 861.945,A -85,B 0,C 180,E1 -24230.06,E2 -24230.06} C_VEL
LIN {X 0,Y 146.477,Z 858.078,A -85,B 0,C 180,E1 -24235.583,E2 -24235.583} C_VEL
LIN {X 0,Y 151.869,Z 851.78,A -85,B 0,C 180,E1 -24242.152,E2 -24242.152} C_VEL
LIN {X 0,Y 157.43,Z 845.37,A -85,B 0,C 180,E1 -24247.06,E2 -24247.06} C_VEL
LIN {X 0,Y 164.139,Z 837.703,A -85,B 0,C 180,E1 -24251.579,E2 -24251.579} C_VEL
LIN {X 0,Y 169.709,Z 831.05,A -85,B 0,C 180,E1 -24254.748,E2 -24254.748} C_VEL
LIN {X 0,Y 175.738,Z 823.499,A -85,B 0,C 180,E1 -24257.716,E2 -24257.716} C_VEL
LIN {X 0,Y 182.257,Z 814.92,A -85,B 0,C 180,E1 -24260.462,E2 -24260.462} C_VEL
LIN {X 0,Y 189.215,Z 805.139,A -85,B 0,C 180,E1 -24262.992,E2 -24262.992} C_VEL
LIN {X 0,Y 195.627,Z 795.356,A -85,B 0,C 180,E1 -24265.07,E2 -24265.07} C_VEL
LIN {X 0,Y 201.51,Z 785.508,A -85,B 0,C 180,E1 -24266.827,E2 -24266.827} C_VEL
LIN {X 0,Y 207.977,Z 773.56,A -85,B 0,C 180,E1 -24268.565,E2 -24268.565} C_VEL
LIN {X 0,Y 213.329,Z 762.63,A -85,B 0,C 180,E1 -24269.856,E2 -24269.856} C_VEL
LIN {X 0,Y 218.715,Z 750.158,A -85,B 0,C 180,E1 -24271.069,E2 -24271.069} C_VEL
LIN {X 0,Y 223.249,Z 737.972,A -85,B 0,C 180,E1 -24272.056,E2 -24272.056} C_VEL
LIN {X 0,Y 227.481,Z 724.774,A -85,B 0,C 180,E1 -24272.89,E2 -24272.89} C_VEL
LIN {X 0,Y 230.894,Z 712.038,A -85,B 0,C 180,E1 -24273.515,E2 -24273.515} C_VEL
LIN {X 0,Y 233.559,Z 699.437,A -85,B 0,C 180,E1 -24274.019,E2 -24274.019} C_VEL
LIN {X 0,Y 235.548,Z 686.833,A -85,B 0,C 180,E1 -24274.42,E2 -24274.42} C_VEL
LIN {X 0,Y 238.706,Z 655.295,A -85,B 0,C 180,E1 -24275.156,E2 -24275.156} C_VEL
LIN {X 0,Y 243.07,Z 607.748,A -85,B 0,C 180,E1 -24276.227,E2 -24276.227} C_VEL
LIN {X 0,Y 239.765,Z 598.653,A -85,B 0,C 180,E1 -24278.788,E2 -24278.788} C_VEL
LIN {X 0,Y 238.027,Z 594.859,A -85,B 0,C 180,E1 -24280.207,E2 -24280.207} C_VEL
LIN {X 0,Y 234.931,Z 589.058,A -85,B 0,C 180,E1 -24282.974,E2 -24282.974} C_VEL
LIN {X 0,Y 232.286,Z 584.408,A -85,B 0,C 180,E1 -24285.774,E2 -24285.774} C_VEL
LIN {X 0,Y 230.836,Z 581.957,A -85,B 0,C 180,E1 -24287.583,E2 -24287.583} C_VEL
LIN {X 0,Y 229.333,Z 579.177,A -85,B 0,C 180,E1 -24289.851,E2 -24289.851} C_VEL
LIN {X 0,Y 227.412,Z 575.53,A -85,B 0,C 180,E1 -24293.919,E2 -24293.919} C_VEL
LIN {X 0,Y 226.861,Z 574.951,A -85,B 0,C 180,E1 -24295.558,E2 -24295.558} C_VEL
LIN {X 0,Y 226.243,Z 573.917,A -85,B 0,C 180,E1 -24300,E2 -24300} C_VEL
LIN {X 0,Y 227.397,Z 575.42,A -85,B 0,C 180,E1 -24306.432,E2 -24306.432} C_VEL
LIN {X 0,Y 229.209,Z 579.073,A -85,B 0,C 180,E1 -24310.377,E2 -24310.377} C_VEL
LIN {X 0,Y 230.011,Z 580.45,A -85,B 0,C 180,E1 -24311.651,E2 -24311.651} C_VEL
LIN {X 0,Y 232.126,Z 584.215,A -85,B 0,C 180,E1 -24314.464,E2 -24314.464} C_VEL
LIN {X 0,Y 234.956,Z 589.027,A -85,B 0,C 180,E1 -24317.459,E2 -24317.459} C_VEL
LIN {X 0,Y 238.631,Z 595.943,A -85,B 0,C 180,E1 -24320.696,E2 -24320.696} C_VEL
LIN {X 0,Y 242.259,Z 603.266,A -85,B 0,C 180,E1 -24323.427,E2 -24323.427} C_VEL
LIN {X 0,Y 249.336,Z 615.384,A -85,B 0,C 180,E1 -24327.715,E2 -24327.715} C_VEL
LIN {X 0,Y 255.49,Z 623.562,A -85,B 0,C 180,E1 -24330.704,E2 -24330.704} C_VEL
LIN {X 0,Y 263.022,Z 631.831,A -85,B 0,C 180,E1 -24333.787,E2 -24333.787} C_VEL
LIN {X 0,Y 280.068,Z 646.599,A -85,B 0,C 180,E1 -24339.317,E2 -24339.317} C_VEL
LIN {X 0,Y 289.116,Z 653.68,A -85,B 0,C 180,E1 -24341.95,E2 -24341.95} C_VEL
LIN {X 0,Y 296.111,Z 659.224,A -85,B 0,C 180,E1 -24344.168,E2 -24344.168} C_VEL
LIN {X 0,Y 301.717,Z 663.498,A -85,B 0,C 180,E1 -24346.067,E2 -24346.067} C_VEL
LIN {X 0,Y 306.639,Z 667.711,A -85,B 0,C 180,E1 -24347.884,E2 -24347.884} C_VEL
LIN {X 0,Y 312.775,Z 672.612,A -85,B 0,C 180,E1 -24350.288,E2 -24350.288} C_VEL
LIN {X 0,Y 318.604,Z 677.407,A -85,B 0,C 180,E1 -24352.722,E2 -24352.722} C_VEL
LIN {X 0,Y 322.239,Z 680.204,A -85,B 0,C 180,E1 -24354.293,E2 -24354.293} C_VEL
LIN {X 0,Y 327.879,Z 684.819,A -85,B 0,C 180,E1 -24356.839,E2 -24356.839} C_VEL
LIN {X 0,Y 331.882,Z 687.893,A -85,B 0,C 180,E1 -24358.74,E2 -24358.74} C_VEL
LIN {X 0,Y 337.029,Z 692.174,A -85,B 0,C 180,E1 -24361.34,E2 -24361.34} C_VEL
LIN {X 0,Y 342.26,Z 695.778,A -85,B 0,C 180,E1 -24364.153,E2 -24364.153} C_VEL
LIN {X 0,Y 346.515,Z 699.356,A -85,B 0,C 180,E1 -24366.698,E2 -24366.698} C_VEL
LIN {X 0,Y 350.549,Z 702.1,A -85,B 0,C 180,E1 -24369.302,E2 -24369.302} C_VEL
LIN {X 0,Y 353.66,Z 704.086,A -85,B 0,C 180,E1 -24371.546,E2 -24371.546} C_VEL
LIN {X 0,Y 356.587,Z 706.748,A -85,B 0,C 180,E1 -24373.983,E2 -24373.983} C_VEL
LIN {X 0,Y 359.328,Z 708.784,A -85,B 0,C 180,E1 -24376.566,E2 -24376.566} C_VEL
LIN {X 0,Y 361.289,Z 710.031,A -85,B 0,C 180,E1 -24378.783,E2 -24378.783} C_VEL
LIN {X 0,Y 363.316,Z 710.904,A -85,B 0,C 180,E1 -24381.475,E2 -24381.475} C_VEL
LIN {X 0,Y 364.522,Z 711.501,A -85,B 0,C 180,E1 -24383.728,E2 -24383.728} C_VEL
LIN {X 0,Y 365.246,Z 711.952,A -85,B 0,C 180,E1 -24385.586,E2 -24385.586} C_VEL
LIN {X 0,Y 365.825,Z 712.054,A -85,B 0,C 180,E1 -24387.798,E2 -24387.798} C_VEL
LIN {X 0,Y 366.037,Z 712.263,A -85,B 0,C 180,E1 -24390,E2 -24390} C_VEL
LIN {X 0,Y 365.774,Z 712.08,A -85,B 0,C 180,E1 -24392.407,E2 -24392.407} C_VEL
LIN {X 0,Y 365.098,Z 711.858,A -85,B 0,C 180,E1 -24394.969,E2 -24394.969} C_VEL
LIN {X 0,Y 364.003,Z 711.223,A -85,B 0,C 180,E1 -24397.297,E2 -24397.297} C_VEL
LIN {X 0,Y 362.252,Z 710.453,A -85,B 0,C 180,E1 -24400.056,E2 -24400.056} C_VEL
LIN {X 0,Y 360.073,Z 709.288,A -85,B 0,C 180,E1 -24402.604,E2 -24402.604} C_VEL
LIN {X 0,Y 357.385,Z 707.396,A -85,B 0,C 180,E1 -24405.295,E2 -24405.295} C_VEL
LIN {X 0,Y 354.371,Z 704.778,A -85,B 0,C 180,E1 -24407.913,E2 -24407.913} C_VEL
LIN {X 0,Y 352.574,Z 703.254,A -85,B 0,C 180,E1 -24409.29,E2 -24409.29} C_VEL
LIN {X 0,Y 348.986,Z 701.107,A -85,B 0,C 180,E1 -24411.726,E2 -24411.726} C_VEL
LIN {X 0,Y 344.796,Z 698.057,A -85,B 0,C 180,E1 -24414.349,E2 -24414.349} C_VEL
LIN {X 0,Y 340.768,Z 694.634,A -85,B 0,C 180,E1 -24416.697,E2 -24416.697} C_VEL
LIN {X 0,Y 337.035,Z 692.125,A -85,B 0,C 180,E1 -24418.659,E2 -24418.659} C_VEL
LIN {X 0,Y 332.013,Z 688.003,A -85,B 0,C 180,E1 -24421.195,E2 -24421.195} C_VEL
LIN {X 0,Y 327.996,Z 684.917,A -85,B 0,C 180,E1 -24423.108,E2 -24423.108} C_VEL
LIN {X 0,Y 322.328,Z 680.299,A -85,B 0,C 180,E1 -24425.667,E2 -24425.667} C_VEL
LIN {X 0,Y 315.474,Z 674.931,A -85,B 0,C 180,E1 -24428.591,E2 -24428.591} C_VEL
LIN {X 0,Y 309.254,Z 669.674,A -85,B 0,C 180,E1 -24431.137,E2 -24431.137} C_VEL
LIN {X 0,Y 303.267,Z 664.89,A -85,B 0,C 180,E1 -24433.38,E2 -24433.38} C_VEL
LIN {X 0,Y 297.241,Z 660.121,A -85,B 0,C 180,E1 -24435.461,E2 -24435.461} C_VEL
LIN {X 0,Y 291.247,Z 655.2,A -85,B 0,C 180,E1 -24437.397,E2 -24437.397} C_VEL
LIN {X 0,Y 284.392,Z 649.992,A -85,B 0,C 180,E1 -24439.441,E2 -24439.441} C_VEL
LIN {X 0,Y 265.959,Z 634.673,A -85,B 0,C 180,E1 -24445.139,E2 -24445.139} C_VEL
LIN {X 0,Y 256.786,Z 625.133,A -85,B 0,C 180,E1 -24448.725,E2 -24448.725} C_VEL
LIN {X 0,Y 249.51,Z 615.658,A -85,B 0,C 180,E1 -24452.192,E2 -24452.192} C_VEL
LIN {X 0,Y 242.34,Z 603.431,A -85,B 0,C 180,E1 -24456.517,E2 -24456.517} C_VEL
LIN {X 0,Y 238.631,Z 595.944,A -85,B 0,C 180,E1 -24459.304,E2 -24459.304} C_VEL
LIN {X 0,Y 234.9,Z 588.962,A -85,B 0,C 180,E1 -24462.591,E2 -24462.591} C_VEL
LIN {X 0,Y 233.148,Z 586.026,A -85,B 0,C 180,E1 -24464.371,E2 -24464.371} C_VEL
LIN {X 0,Y 231.17,Z 582.488,A -85,B 0,C 180,E1 -24466.731,E2 -24466.731} C_VEL
LIN {X 0,Y 229.346,Z 579.238,A -85,B 0,C 180,E1 -24469.406,E2 -24469.406} C_VEL
LIN {X 0,Y 227.393,Z 575.459,A -85,B 0,C 180,E1 -24473.568,E2 -24473.568} C_VEL
LIN {X 0,Y 226.748,Z 574.834,A -85,B 0,C 180,E1 -24475.556,E2 -24475.556} C_VEL
LIN {X 0,Y 226.24,Z 573.944,A -85,B 0,C 180,E1 -24480,E2 -24480} C_VEL
LIN {X 0,Y 227.412,Z 575.477,A -85,B 0,C 180,E1 -24486.067,E2 -24486.067} C_VEL
LIN {X 0,Y 229.184,Z 579.046,A -85,B 0,C 180,E1 -24489.921,E2 -24489.921} C_VEL
LIN {X 0,Y 229.93,Z 580.208,A -85,B 0,C 180,E1 -24491.097,E2 -24491.097} C_VEL
LIN {X 0,Y 232.111,Z 584.089,A -85,B 0,C 180,E1 -24494.018,E2 -24494.018} C_VEL
LIN {X 0,Y 235.046,Z 589.256,A -85,B 0,C 180,E1 -24497.137,E2 -24497.137} C_VEL
LIN {X 0,Y 238.087,Z 594.989,A -85,B 0,C 180,E1 -24499.844,E2 -24499.844} C_VEL
LIN {X 0,Y 239.767,Z 598.642,A -85,B 0,C 180,E1 -24501.212,E2 -24501.212} C_VEL
LIN {X 0,Y 243.013,Z 607.535,A -85,B 0,C 180,E1 -24503.728,E2 -24503.728} C_VEL
LIN {X 0,Y 241.685,Z 623.078,A -85,B 0,C 180,E1 -24504.131,E2 -24504.131} C_VEL
LIN {X 0,Y 235.859,Z 684.673,A -85,B 0,C 180,E1 -24505.534,E2 -24505.534} C_VEL
LIN {X 0,Y 233.903,Z 697.438,A -85,B 0,C 180,E1 -24505.908,E2 -24505.908} C_VEL
LIN {X 0,Y 231.243,Z 710.506,A -85,B 0,C 180,E1 -24506.414,E2 -24506.414} C_VEL
LIN {X 0,Y 228.186,Z 722.306,A -85,B 0,C 180,E1 -24506.971,E2 -24506.971} C_VEL
LIN {X 0,Y 224.301,Z 734.896,A -85,B 0,C 180,E1 -24507.732,E2 -24507.732} C_VEL
LIN {X 0,Y 220.176,Z 746.437,A -85,B 0,C 180,E1 -24508.607,E2 -24508.607} C_VEL
LIN {X 0,Y 215.368,Z 758.134,A -85,B 0,C 180,E1 -24509.678,E2 -24509.678} C_VEL
LIN {X 0,Y 209.312,Z 770.952,A -85,B 0,C 180,E1 -24511.109,E2 -24511.109} C_VEL
LIN {X 0,Y 203.458,Z 782.08,A -85,B 0,C 180,E1 -24512.653,E2 -24512.653} C_VEL
LIN {X 0,Y 197.079,Z 792.911,A -85,B 0,C 180,E1 -24514.448,E2 -24514.448} C_VEL
LIN {X 0,Y 190.433,Z 803.366,A -85,B 0,C 180,E1 -24516.614,E2 -24516.614} C_VEL
LIN {X 0,Y 184.522,Z 811.789,A -85,B 0,C 180,E1 -24518.668,E2 -24518.668} C_VEL
LIN {X 0,Y 177.862,Z 820.743,A -85,B 0,C 180,E1 -24521.345,E2 -24521.345} C_VEL
LIN {X 0,Y 171.514,Z 828.776,A -85,B 0,C 180,E1 -24524.288,E2 -24524.288} C_VEL
LIN {X 0,Y 165.968,Z 835.598,A -85,B 0,C 180,E1 -24527.35,E2 -24527.35} C_VEL
LIN {X 0,Y 160.658,Z 841.736,A -85,B 0,C 180,E1 -24530.633,E2 -24530.633} C_VEL
LIN {X 0,Y 154.394,Z 848.832,A -85,B 0,C 180,E1 -24535.469,E2 -24535.469} C_VEL
LIN {X 0,Y 149.462,Z 854.453,A -85,B 0,C 180,E1 -24540.415,E2 -24540.415} C_VEL
LIN {X 0,Y 146.475,Z 858.078,A -85,B 0,C 180,E1 -24544.417,E2 -24544.417} C_VEL
LIN {X 0,Y 143.427,Z 861.945,A -85,B 0,C 180,E1 -24549.94,E2 -24549.94} C_VEL
LIN {X 0,Y 141.392,Z 864.812,A -85,B 0,C 180,E1 -24555.61,E2 -24555.61} C_VEL
LIN {X 0,Y 140.853,Z 865.959,A -85,B 0,C 180,E1 -24558.488,E2 -24558.488} C_VEL
LIN {X 0,Y 140.44,Z 867.406,A -85,B 0,C 180,E1 -24564.256,E2 -24564.256} C_VEL
LIN {X 0,Y 140.6,Z 867.895,A -85,B 0,C 180,E1 -24570,E2 -24570} C_VEL
LIN {X 0,Y 140.44,Z 867.406,A -85,B 0,C 180,E1 -24575.744,E2 -24575.744} C_VEL
LIN {X 0,Y 140.58,Z 866.527,A -85,B 0,C 180,E1 -24579.356,E2 -24579.356} C_VEL
LIN {X 0,Y 140.199,Z 865.87,A -85,B 0,C 180,E1 -24581.743,E2 -24581.743} C_VEL
LIN {X 0,Y 138.207,Z 864.34,A -85,B 0,C 180,E1 -24585.694,E2 -24585.694} C_VEL
LIN {X 0,Y 136.872,Z 862.874,A -85,B 0,C 180,E1 -24588.911,E2 -24588.911} C_VEL
LIN {X 0,Y 136.894,Z 861.594,A -85,B 0,C 180,E1 -24591.337,E2 -24591.337} C_VEL
LIN {X 0,Y 137.209,Z 861.121,A -85,B 0,C 180,E1 -24592.131,E2 -24592.131} C_VEL
LIN {X 0,Y 140.994,Z 856.806,A -85,B 0,C 180,E1 -24598.263,E2 -24598.263} C_VEL
LIN {X 0,Y 145.798,Z 851.566,A -85,B 0,C 180,E1 -24603.665,E2 -24603.665} C_VEL
LIN {X 0,Y 151.724,Z 845.156,A -85,B 0,C 180,E1 -24608.706,E2 -24608.706} C_VEL
LIN {X 0,Y 158.813,Z 837.49,A -85,B 0,C 180,E1 -24613.307,E2 -24613.307} C_VEL
LIN {X 0,Y 164.633,Z 830.835,A -85,B 0,C 180,E1 -24616.527,E2 -24616.527} C_VEL
LIN {X 0,Y 170.965,Z 823.286,A -85,B 0,C 180,E1 -24619.506,E2 -24619.506} C_VEL
LIN {X 0,Y 177.748,Z 814.707,A -85,B 0,C 180,E1 -24622.257,E2 -24622.257} C_VEL
LIN {X 0,Y 184.994,Z 804.927,A -85,B 0,C 180,E1 -24624.763,E2 -24624.763} C_VEL
LIN {X 0,Y 191.475,Z 795.333,A -85,B 0,C 180,E1 -24626.8,E2 -24626.8} C_VEL
LIN {X 0,Y 197.682,Z 785.296,A -85,B 0,C 180,E1 -24628.564,E2 -24628.564} C_VEL
LIN {X 0,Y 204.35,Z 773.35,A -85,B 0,C 180,E1 -24630.271,E2 -24630.271} C_VEL
LIN {X 0,Y 209.83,Z 762.419,A -85,B 0,C 180,E1 -24631.545,E2 -24631.545} C_VEL
LIN {X 0,Y 215.328,Z 749.945,A -85,B 0,C 180,E1 -24632.744,E2 -24632.744} C_VEL
LIN {X 0,Y 220.005,Z 737.762,A -85,B 0,C 180,E1 -24633.693,E2 -24633.693} C_VEL
LIN {X 0,Y 224.334,Z 724.564,A -85,B 0,C 180,E1 -24634.505,E2 -24634.505} C_VEL
LIN {X 0,Y 227.817,Z 711.829,A -85,B 0,C 180,E1 -24635.113,E2 -24635.113} C_VEL
LIN {X 0,Y 230.537,Z 699.228,A -85,B 0,C 180,E1 -24635.606,E2 -24635.606} C_VEL
LIN {X 0,Y 232.609,Z 686.331,A -85,B 0,C 180,E1 -24636.004,E2 -24636.004} C_VEL
LIN {X 0,Y 235.813,Z 655.085,A -85,B 0,C 180,E1 -24636.72,E2 -24636.72} C_VEL
LIN {X 0,Y 239.92,Z 610.974,A -85,B 0,C 180,E1 -24637.729,E2 -24637.729} C_VEL
LIN {X 0,Y 237.293,Z 603.537,A -85,B 0,C 180,E1 -24639.943,E2 -24639.943} C_VEL
LIN {X 0,Y 235.225,Z 599.075,A -85,B 0,C 180,E1 -24641.772,E2 -24641.772} C_VEL
LIN {X 0,Y 232.219,Z 593.367,A -85,B 0,C 180,E1 -24644.782,E2 -24644.782} C_VEL
LIN {X 0,Y 229.797,Z 589.026,A -85,B 0,C 180,E1 -24647.75,E2 -24647.75} C_VEL
LIN {X 0,Y 228.25,Z 586.084,A -85,B 0,C 180,E1 -24650.158,E2 -24650.158} C_VEL
LIN {X 0,Y 226.287,Z 582.199,A -85,B 0,C 180,E1 -24654.653,E2 -24654.653} C_VEL
LIN {X 0,Y 225.377,Z 580.969,A -85,B 0,C 180,E1 -24660,E2 -24660} C_VEL
LIN {X 0,Y 226.405,Z 582.413,A -85,B 0,C 180,E1 -24666.125,E2 -24666.125} C_VEL
LIN {X 0,Y 228.209,Z 586.077,A -85,B 0,C 180,E1 -24670.199,E2 -24670.199} C_VEL
LIN {X 0,Y 230.467,Z 590.22,A -85,B 0,C 180,E1 -24673.557,E2 -24673.557} C_VEL
LIN {X 0,Y 233.456,Z 595.621,A -85,B 0,C 180,E1 -24676.936,E2 -24676.936} C_VEL
LIN {X 0,Y 237.132,Z 602.877,A -85,B 0,C 180,E1 -24680.311,E2 -24680.311} C_VEL
LIN {X 0,Y 246.974,Z 621.391,A -85,B 0,C 180,E1 -24687.025,E2 -24687.025} C_VEL
LIN {X 0,Y 253.069,Z 629.698,A -85,B 0,C 180,E1 -24690.104,E2 -24690.104} C_VEL
LIN {X 0,Y 260.999,Z 638.478,A -85,B 0,C 180,E1 -24693.44,E2 -24693.44} C_VEL
LIN {X 0,Y 277.387,Z 652.853,A -85,B 0,C 180,E1 -24698.885,E2 -24698.885} C_VEL
LIN {X 0,Y 287.681,Z 660.77,A -85,B 0,C 180,E1 -24701.854,E2 -24701.854} C_VEL
LIN {X 0,Y 294.843,Z 666.457,A -85,B 0,C 180,E1 -24704.114,E2 -24704.114} C_VEL
LIN {X 0,Y 300.836,Z 671.082,A -85,B 0,C 180,E1 -24706.127,E2 -24706.127} C_VEL
LIN {X 0,Y 306.868,Z 675.981,A -85,B 0,C 180,E1 -24708.343,E2 -24708.343} C_VEL
LIN {X 0,Y 312.059,Z 680.19,A -85,B 0,C 180,E1 -24710.407,E2 -24710.407} C_VEL
LIN {X 0,Y 317.974,Z 684.869,A -85,B 0,C 180,E1 -24712.871,E2 -24712.871} C_VEL
LIN {X 0,Y 321.943,Z 688.117,A -85,B 0,C 180,E1 -24714.595,E2 -24714.595} C_VEL
LIN {X 0,Y 327.545,Z 692.411,A -85,B 0,C 180,E1 -24717.119,E2 -24717.119} C_VEL
LIN {X 0,Y 331.389,Z 695.509,A -85,B 0,C 180,E1 -24718.966,E2 -24718.966} C_VEL
LIN {X 0,Y 336.202,Z 699.43,A -85,B 0,C 180,E1 -24721.398,E2 -24721.398} C_VEL
LIN {X 0,Y 341.118,Z 702.791,A -85,B 0,C 180,E1 -24724.031,E2 -24724.031} C_VEL
LIN {X 0,Y 345.491,Z 706.385,A -85,B 0,C 180,E1 -24726.625,E2 -24726.625} C_VEL
LIN {X 0,Y 349.575,Z 709.102,A -85,B 0,C 180,E1 -24729.241,E2 -24729.241} C_VEL
LIN {X 0,Y 352.568,Z 711.057,A -85,B 0,C 180,E1 -24731.402,E2 -24731.402} C_VEL
LIN {X 0,Y 355.656,Z 713.79,A -85,B 0,C 180,E1 -24733.94,E2 -24733.94} C_VEL
LIN {X 0,Y 358.249,Z 715.726,A -85,B 0,C 180,E1 -24736.384,E2 -24736.384} C_VEL
LIN {X 0,Y 360.393,Z 717.072,A -85,B 0,C 180,E1 -24738.755,E2 -24738.755} C_VEL
LIN {X 0,Y 362.437,Z 717.925,A -85,B 0,C 180,E1 -24741.465,E2 -24741.465} C_VEL
LIN {X 0,Y 363.648,Z 718.547,A -85,B 0,C 180,E1 -24743.713,E2 -24743.713} C_VEL
LIN {X 0,Y 364.375,Z 718.997,A -85,B 0,C 180,E1 -24745.575,E2 -24745.575} C_VEL
LIN {X 0,Y 364.956,Z 719.102,A -85,B 0,C 180,E1 -24747.793,E2 -24747.793} C_VEL
LIN {X 0,Y 365.172,Z 719.309,A -85,B 0,C 180,E1 -24750,E2 -24750} C_VEL
LIN {X 0,Y 364.956,Z 719.101,A -85,B 0,C 180,E1 -24752.207,E2 -24752.207} C_VEL
LIN {X 0,Y 364.379,Z 718.968,A -85,B 0,C 180,E1 -24754.425,E2 -24754.425} C_VEL
LIN {X 0,Y 363.123,Z 718.255,A -85,B 0,C 180,E1 -24757.315,E2 -24757.315} C_VEL
LIN {X 0,Y 361.36,Z 717.494,A -85,B 0,C 180,E1 -24760.081,E2 -24760.081} C_VEL
LIN {X 0,Y 359.166,Z 716.33,A -85,B 0,C 180,E1 -24762.636,E2 -24762.636} C_VEL
LIN {X 0,Y 356.354,Z 714.378,A -85,B 0,C 180,E1 -24765.419,E2 -24765.419} C_VEL
LIN {X 0,Y 353.29,Z 711.74,A -85,B 0,C 180,E1 -24768.054,E2 -24768.054} C_VEL
LIN {X 0,Y 351.402,Z 710.175,A -85,B 0,C 180,E1 -24769.496,E2 -24769.496} C_VEL
LIN {X 0,Y 347.763,Z 707.983,A -85,B 0,C 180,E1 -24771.94,E2 -24771.94} C_VEL
LIN {X 0,Y 343.58,Z 704.974,A -85,B 0,C 180,E1 -24774.524,E2 -24774.524} C_VEL
LIN {X 0,Y 339.662,Z 701.621,A -85,B 0,C 180,E1 -24776.791,E2 -24776.791} C_VEL
LIN {X 0,Y 335.649,Z 698.951,A -85,B 0,C 180,E1 -24778.897,E2 -24778.897} C_VEL
LIN {X 0,Y 330.705,Z 694.956,A -85,B 0,C 180,E1 -24781.37,E2 -24781.37} C_VEL
LIN {X 0,Y 326.825,Z 691.897,A -85,B 0,C 180,E1 -24783.205,E2 -24783.205} C_VEL
LIN {X 0,Y 321.289,Z 687.576,A -85,B 0,C 180,E1 -24785.689,E2 -24785.689} C_VEL
LIN {X 0,Y 316.307,Z 683.629,A -85,B 0,C 180,E1 -24787.828,E2 -24787.828} C_VEL
LIN {X 0,Y 309.99,Z 678.364,A -85,B 0,C 180,E1 -24790.437,E2 -24790.437} C_VEL
LIN {X 0,Y 303.107,Z 673.01,A -85,B 0,C 180,E1 -24793.067,E2 -24793.067} C_VEL
LIN {X 0,Y 297.404,Z 668.363,A -85,B 0,C 180,E1 -24795.054,E2 -24795.054} C_VEL
LIN {X 0,Y 290.924,Z 663.33,A -85,B 0,C 180,E1 -24797.141,E2 -24797.141} C_VEL
LIN {X 0,Y 283.907,Z 657.944,A -85,B 0,C 180,E1 -24799.24,E2 -24799.24} C_VEL
LIN {X 0,Y 264.37,Z 641.808,A -85,B 0,C 180,E1 -24805.304,E2 -24805.304} C_VEL
LIN {X 0,Y 254.542,Z 631.486,A -85,B 0,C 180,E1 -24809.227,E2 -24809.227} C_VEL
LIN {X 0,Y 247.403,Z 622.047,A -85,B 0,C 180,E1 -24812.738,E2 -24812.738} C_VEL
LIN {X 0,Y 240.41,Z 609.835,A -85,B 0,C 180,E1 -24817.119,E2 -24817.119} C_VEL
LIN {X 0,Y 236.809,Z 602.221,A -85,B 0,C 180,E1 -24819.962,E2 -24819.962} C_VEL
LIN {X 0,Y 233.149,Z 595.133,A -85,B 0,C 180,E1 -24823.369,E2 -24823.369} C_VEL
LIN {X 0,Y 231.317,Z 591.937,A -85,B 0,C 180,E1 -24825.372,E2 -24825.372} C_VEL
LIN {X 0,Y 229.735,Z 588.981,A -85,B 0,C 180,E1 -24827.411,E2 -24827.411} C_VEL
LIN {X 0,Y 228.21,Z 586.072,A -85,B 0,C 180,E1 -24829.801,E2 -24829.801} C_VEL
LIN {X 0,Y 226.304,Z 582.156,A -85,B 0,C 180,E1 -24834.208,E2 -24834.208} C_VEL
LIN {X 0,Y 225.374,Z 580.997,A -85,B 0,C 180,E1 -24840,E2 -24840} C_VEL
LIN {X 0,Y 226.441,Z 582.46,A -85,B 0,C 180,E1 -24845.812,E2 -24845.812} C_VEL
LIN {X 0,Y 228.117,Z 585.968,A -85,B 0,C 180,E1 -24849.631,E2 -24849.631} C_VEL
LIN {X 0,Y 228.98,Z 587.561,A -85,B 0,C 180,E1 -24851.06,E2 -24851.06} C_VEL
LIN {X 0,Y 230.865,Z 590.961,A -85,B 0,C 180,E1 -24853.646,E2 -24853.646} C_VEL
LIN {X 0,Y 233.382,Z 595.579,A -85,B 0,C 180,E1 -24856.455,E2 -24856.455} C_VEL
LIN {X 0,Y 236.257,Z 601.201,A -85,B 0,C 180,E1 -24859.157,E2 -24859.157} C_VEL
LIN {X 0,Y 237.91,Z 605.172,A -85,B 0,C 180,E1 -24860.593,E2 -24860.593} C_VEL
LIN {X 0,Y 239.958,Z 611.059,A -85,B 0,C 180,E1 -24862.299,E2 -24862.299} C_VEL
LIN {X 0,Y 232.764,Z 685.39,A -85,B 0,C 180,E1 -24863.98,E2 -24863.98} C_VEL
LIN {X 0,Y 230.546,Z 699.228,A -85,B 0,C 180,E1 -24864.399,E2 -24864.399} C_VEL
LIN {X 0,Y 227.238,Z 714.124,A -85,B 0,C 180,E1 -24864.967,E2 -24864.967} C_VEL
LIN {X 0,Y 222.158,Z 731.61,A -85,B 0,C 180,E1 -24865.894,E2 -24865.894} C_VEL
LIN {X 0,Y 217.142,Z 745.519,A -85,B 0,C 180,E1 -24866.895,E2 -24866.895} C_VEL
LIN {X 0,Y 211.92,Z 757.923,A -85,B 0,C 180,E1 -24867.999,E2 -24867.999} C_VEL
LIN {X 0,Y 205.712,Z 770.741,A -85,B 0,C 180,E1 -24869.406,E2 -24869.406} C_VEL
LIN {X 0,Y 199.668,Z 781.868,A -85,B 0,C 180,E1 -24870.914,E2 -24870.914} C_VEL
LIN {X 0,Y 193.115,Z 792.699,A -85,B 0,C 180,E1 -24872.695,E2 -24872.695} C_VEL
LIN {X 0,Y 187.466,Z 801.379,A -85,B 0,C 180,E1 -24874.437,E2 -24874.437} C_VEL
LIN {X 0,Y 180.123,Z 811.577,A -85,B 0,C 180,E1 -24876.885,E2 -24876.885} C_VEL
LIN {X 0,Y 173.185,Z 820.53,A -85,B 0,C 180,E1 -24879.554,E2 -24879.554} C_VEL
LIN {X 0,Y 166.736,Z 828.332,A -85,B 0,C 180,E1 -24882.408,E2 -24882.408} C_VEL
LIN {X 0,Y 160.757,Z 835.386,A -85,B 0,C 180,E1 -24885.615,E2 -24885.615} C_VEL
LIN {X 0,Y 155.135,Z 841.523,A -85,B 0,C 180,E1 -24888.938,E2 -24888.938} C_VEL
LIN {X 0,Y 149.469,Z 847.609,A -85,B 0,C 180,E1 -24893.067,E2 -24893.067} C_VEL
LIN {X 0,Y 144.491,Z 852.951,A -85,B 0,C 180,E1 -24897.655,E2 -24897.655} C_VEL
LIN {X 0,Y 140.005,Z 857.865,A -85,B 0,C 180,E1 -24903.142,E2 -24903.142} C_VEL
LIN {X 0,Y 136.702,Z 861.733,A -85,B 0,C 180,E1 -24908.908,E2 -24908.908} C_VEL
LIN {X 0,Y 134.448,Z 864.6,A -85,B 0,C 180,E1 -24914.849,E2 -24914.849} C_VEL
LIN {X 0,Y 133.478,Z 866.508,A -85,B 0,C 180,E1 -24920.912,E2 -24920.912} C_VEL
LIN {X 0,Y 133.347,Z 867.196,A -85,B 0,C 180,E1 -24923.949,E2 -24923.949} C_VEL
LIN {X 0,Y 133.502,Z 867.685,A -85,B 0,C 180,E1 -24930,E2 -24930} C_VEL
LIN {X 0,Y 133.347,Z 867.196,A -85,B 0,C 180,E1 -24936.051,E2 -24936.051} C_VEL
LIN {X 0,Y 133.83,Z 865.747,A -85,B 0,C 180,E1 -24942.125,E2 -24942.125} C_VEL
LIN {X 0,Y 135.436,Z 863.342,A -85,B 0,C 180,E1 -24948.14,E2 -24948.14} C_VEL
LIN {X 0,Y 137.209,Z 861.121,A -85,B 0,C 180,E1 -24952.131,E2 -24952.131} C_VEL
LIN {X 0,Y 137.84,Z 859.691,A -85,B 0,C 180,E1 -24954.502,E2 -24954.502} C_VEL
LIN {X 0,Y 137.498,Z 857.07,A -85,B 0,C 180,E1 -24958.482,E2 -24958.482} C_VEL
LIN {X 0,Y 137.495,Z 854.711,A -85,B 0,C 180,E1 -24961.653,E2 -24961.653} C_VEL
LIN {X 0,Y 138.513,Z 852.735,A -85,B 0,C 180,E1 -24963.932,E2 -24963.932} C_VEL
LIN {X 0,Y 139.152,Z 852.027,A -85,B 0,C 180,E1 -24964.647,E2 -24964.647} C_VEL
LIN {X 0,Y 146.168,Z 844.943,A -85,B 0,C 180,E1 -24970.473,E2 -24970.473} C_VEL
LIN {X 0,Y 153.649,Z 837.277,A -85,B 0,C 180,E1 -24975.15,E2 -24975.15} C_VEL
LIN {X 0,Y 159.765,Z 830.623,A -85,B 0,C 180,E1 -24978.401,E2 -24978.401} C_VEL
LIN {X 0,Y 166.385,Z 823.073,A -85,B 0,C 180,E1 -24981.39,E2 -24981.39} C_VEL
LIN {X 0,Y 173.429,Z 814.494,A -85,B 0,C 180,E1 -24984.141,E2 -24984.141} C_VEL
LIN {X 0,Y 180.959,Z 804.716,A -85,B 0,C 180,E1 -24986.615,E2 -24986.615} C_VEL
LIN {X 0,Y 187.495,Z 795.314,A -85,B 0,C 180,E1 -24988.608,E2 -24988.608} C_VEL
LIN {X 0,Y 194.036,Z 785.084,A -85,B 0,C 180,E1 -24990.373,E2 -24990.373} C_VEL
LIN {X 0,Y 200.903,Z 773.139,A -85,B 0,C 180,E1 -24992.04,E2 -24992.04} C_VEL
LIN {X 0,Y 206.532,Z 762.209,A -85,B 0,C 180,E1 -24993.282,E2 -24993.282} C_VEL
LIN {X 0,Y 212.158,Z 749.735,A -85,B 0,C 180,E1 -24994.455,E2 -24994.455} C_VEL
LIN {X 0,Y 216.957,Z 737.552,A -85,B 0,C 180,E1 -24995.371,E2 -24995.371} C_VEL
LIN {X 0,Y 221.364,Z 724.354,A -85,B 0,C 180,E1 -24996.168,E2 -24996.168} C_VEL
LIN {X 0,Y 224.908,Z 711.618,A -85,B 0,C 180,E1 -24996.762,E2 -24996.762} C_VEL
LIN {X 0,Y 227.688,Z 699.017,A -85,B 0,C 180,E1 -24997.239,E2 -24997.239} C_VEL
LIN {X 0,Y 229.824,Z 686.022,A -85,B 0,C 180,E1 -24997.625,E2 -24997.625} C_VEL
LIN {X 0,Y 233.304,Z 652.788,A -85,B 0,C 180,E1 -24998.367,E2 -24998.367} C_VEL
LIN {X 0,Y 236.993,Z 614.524,A -85,B 0,C 180,E1 -24999.21,E2 -24999.21} C_VEL
LIN {X 0,Y 234.815,Z 608.153,A -85,B 0,C 180,E1 -25001.22,E2 -25001.22} C_VEL
LIN {X 0,Y 231.819,Z 602.013,A -85,B 0,C 180,E1 -25004.166,E2 -25004.166} C_VEL
LIN {X 0,Y 228.759,Z 596.101,A -85,B 0,C 180,E1 -25007.919,E2 -25007.919} C_VEL
LIN {X 0,Y 227.066,Z 592.886,A -85,B 0,C 180,E1 -25010.648,E2 -25010.648} C_VEL
LIN {X 0,Y 225.419,Z 589.302,A -85,B 0,C 180,E1 -25014.633,E2 -25014.633} C_VEL
LIN {X 0,Y 224.511,Z 588.021,A -85,B 0,C 180,E1 -25020,E2 -25020} C_VEL
LIN {X 0,Y 225.423,Z 589.365,A -85,B 0,C 180,E1 -25025.815,E2 -25025.815} C_VEL
LIN {X 0,Y 227.515,Z 593.752,A -85,B 0,C 180,E1 -25030.568,E2 -25030.568} C_VEL
LIN {X 0,Y 229.458,Z 597.614,A -85,B 0,C 180,E1 -25033.477,E2 -25033.477} C_VEL
LIN {X 0,Y 231.888,Z 602.094,A -85,B 0,C 180,E1 -25036.318,E2 -25036.318} C_VEL
LIN {X 0,Y 235.244,Z 609,A -85,B 0,C 180,E1 -25039.574,E2 -25039.574} C_VEL
LIN {X 0,Y 244.654,Z 627.396,A -85,B 0,C 180,E1 -25046.324,E2 -25046.324} C_VEL
LIN {X 0,Y 250.959,Z 636.142,A -85,B 0,C 180,E1 -25049.625,E2 -25049.625} C_VEL
LIN {X 0,Y 258.356,Z 644.532,A -85,B 0,C 180,E1 -25052.842,E2 -25052.842} C_VEL
LIN {X 0,Y 275.015,Z 659.327,A -85,B 0,C 180,E1 -25058.532,E2 -25058.532} C_VEL
LIN {X 0,Y 285.997,Z 667.7,A -85,B 0,C 180,E1 -25061.683,E2 -25061.683} C_VEL
LIN {X 0,Y 294.14,Z 674.055,A -85,B 0,C 180,E1 -25064.231,E2 -25064.231} C_VEL
LIN {X 0,Y 300.331,Z 678.995,A -85,B 0,C 180,E1 -25066.365,E2 -25066.365} C_VEL
LIN {X 0,Y 306.825,Z 684.016,A -85,B 0,C 180,E1 -25068.779,E2 -25068.779} C_VEL
LIN {X 0,Y 313.66,Z 689.669,A -85,B 0,C 180,E1 -25071.517,E2 -25071.517} C_VEL
LIN {X 0,Y 319.121,Z 693.833,A -85,B 0,C 180,E1 -25073.805,E2 -25073.805} C_VEL
LIN {X 0,Y 324.898,Z 698.427,A -85,B 0,C 180,E1 -25076.369,E2 -25076.369} C_VEL
LIN {X 0,Y 329.251,Z 701.733,A -85,B 0,C 180,E1 -25078.408,E2 -25078.408} C_VEL
LIN {X 0,Y 334.155,Z 705.774,A -85,B 0,C 180,E1 -25080.844,E2 -25080.844} C_VEL
LIN {X 0,Y 339.561,Z 709.433,A -85,B 0,C 180,E1 -25083.697,E2 -25083.697} C_VEL
LIN {X 0,Y 343.845,Z 713.022,A -85,B 0,C 180,E1 -25086.195,E2 -25086.195} C_VEL
LIN {X 0,Y 348.177,Z 715.931,A -85,B 0,C 180,E1 -25088.953,E2 -25088.953} C_VEL
LIN {X 0,Y 351.404,Z 717.961,A -85,B 0,C 180,E1 -25091.206,E2 -25091.206} C_VEL
LIN {X 0,Y 354.697,Z 720.84,A -85,B 0,C 180,E1 -25093.895,E2 -25093.895} C_VEL
LIN {X 0,Y 357.469,Z 722.887,A -85,B 0,C 180,E1 -25096.516,E2 -25096.516} C_VEL
LIN {X 0,Y 359.91,Z 724.299,A -85,B 0,C 180,E1 -25099.266,E2 -25099.266} C_VEL
LIN {X 0,Y 361.959,Z 725.146,A -85,B 0,C 180,E1 -25102.189,E2 -25102.189} C_VEL
LIN {X 0,Y 363.077,Z 725.773,A -85,B 0,C 180,E1 -25104.446,E2 -25104.446} C_VEL
LIN {X 0,Y 363.857,Z 726.162,A -85,B 0,C 180,E1 -25106.678,E2 -25106.678} C_VEL
LIN {X 0,Y 364.199,Z 726.295,A -85,B 0,C 180,E1 -25108.894,E2 -25108.894} C_VEL
LIN {X 0,Y 364.194,Z 726.295,A -85,B 0,C 180,E1 -25111.106,E2 -25111.106} C_VEL
LIN {X 0,Y 363.849,Z 726.188,A -85,B 0,C 180,E1 -25113.322,E2 -25113.322} C_VEL
LIN {X 0,Y 362.916,Z 725.671,A -85,B 0,C 180,E1 -25115.928,E2 -25115.928} C_VEL
LIN {X 0,Y 361.516,Z 724.976,A -85,B 0,C 180,E1 -25118.555,E2 -25118.555} C_VEL
LIN {X 0,Y 359.482,Z 724.076,A -85,B 0,C 180,E1 -25121.274,E2 -25121.274} C_VEL
LIN {X 0,Y 356.87,Z 722.49,A -85,B 0,C 180,E1 -25124.076,E2 -25124.076} C_VEL
LIN {X 0,Y 353.891,Z 720.204,A -85,B 0,C 180,E1 -25126.787,E2 -25126.787} C_VEL
LIN {X 0,Y 350.833,Z 717.387,A -85,B 0,C 180,E1 -25129.245,E2 -25129.245} C_VEL
LIN {X 0,Y 347.034,Z 715.188,A -85,B 0,C 180,E1 -25131.814,E2 -25131.814} C_VEL
LIN {X 0,Y 342.635,Z 712.123,A -85,B 0,C 180,E1 -25134.512,E2 -25134.512} C_VEL
LIN {X 0,Y 338.105,Z 708.381,A -85,B 0,C 180,E1 -25137.114,E2 -25137.114} C_VEL
LIN {X 0,Y 333.744,Z 705.414,A -85,B 0,C 180,E1 -25139.369,E2 -25139.369} C_VEL
LIN {X 0,Y 328.752,Z 701.312,A -85,B 0,C 180,E1 -25141.836,E2 -25141.836} C_VEL
LIN {X 0,Y 322.537,Z 696.67,A -85,B 0,C 180,E1 -25144.679,E2 -25144.679} C_VEL
LIN {X 0,Y 316.462,Z 691.742,A -85,B 0,C 180,E1 -25147.321,E2 -25147.321} C_VEL
LIN {X 0,Y 310.162,Z 686.805,A -85,B 0,C 180,E1 -25149.902,E2 -25149.902} C_VEL
LIN {X 0,Y 304.446,Z 682.237,A -85,B 0,C 180,E1 -25152.125,E2 -25152.125} C_VEL
LIN {X 0,Y 298.225,Z 677.174,A -85,B 0,C 180,E1 -25154.389,E2 -25154.389} C_VEL
LIN {X 0,Y 291.028,Z 671.722,A -85,B 0,C 180,E1 -25156.764,E2 -25156.764} C_VEL
LIN {X 0,Y 284.203,Z 666.411,A -85,B 0,C 180,E1 -25158.822,E2 -25158.822} C_VEL
LIN {X 0,Y 270.277,Z 655.502,A -85,B 0,C 180,E1 -25162.923,E2 -25162.923} C_VEL
LIN {X 0,Y 254.494,Z 640.495,A -85,B 0,C 180,E1 -25168.759,E2 -25168.759} C_VEL
LIN {X 0,Y 245.249,Z 628.336,A -85,B 0,C 180,E1 -25173.333,E2 -25173.333} C_VEL
LIN {X 0,Y 238.273,Z 615.743,A -85,B 0,C 180,E1 -25177.91,E2 -25177.91} C_VEL
LIN {X 0,Y 234.844,Z 608.176,A -85,B 0,C 180,E1 -25180.781,E2 -25180.781} C_VEL
LIN {X 0,Y 231.414,Z 601.197,A -85,B 0,C 180,E1 -25184.195,E2 -25184.195} C_VEL
LIN {X 0,Y 228.516,Z 595.74,A -85,B 0,C 180,E1 -25187.84,E2 -25187.84} C_VEL
LIN {X 0,Y 227.085,Z 592.904,A -85,B 0,C 180,E1 -25190.2,E2 -25190.2} C_VEL
LIN {X 0,Y 225.288,Z 589.12,A -85,B 0,C 180,E1 -25194.63,E2 -25194.63} C_VEL
LIN {X 0,Y 224.509,Z 588.035,A -85,B 0,C 180,E1 -25200,E2 -25200} C_VEL
LIN {X 0,Y 225.45,Z 589.418,A -85,B 0,C 180,E1 -25205.484,E2 -25205.484} C_VEL
LIN {X 0,Y 227.561,Z 593.832,A -85,B 0,C 180,E1 -25210.229,E2 -25210.229} C_VEL
LIN {X 0,Y 229.463,Z 597.528,A -85,B 0,C 180,E1 -25213.055,E2 -25213.055} C_VEL
LIN {X 0,Y 231.66,Z 601.734,A -85,B 0,C 180,E1 -25215.666,E2 -25215.666} C_VEL
LIN {X 0,Y 234.43,Z 607.387,A -85,B 0,C 180,E1 -25218.433,E2 -25218.433} C_VEL
LIN {X 0,Y 235.986,Z 611.39,A -85,B 0,C 180,E1 -25219.873,E2 -25219.873} C_VEL
LIN {X 0,Y 236.991,Z 614.538,A -85,B 0,C 180,E1 -25220.79,E2 -25220.79} C_VEL
LIN {X 0,Y 229.974,Z 685.177,A -85,B 0,C 180,E1 -25222.365,E2 -25222.365} C_VEL
LIN {X 0,Y 227.693,Z 699.018,A -85,B 0,C 180,E1 -25222.765,E2 -25222.765} C_VEL
LIN {X 0,Y 224.523,Z 713.149,A -85,B 0,C 180,E1 -25223.293,E2 -25223.293} C_VEL
LIN {X 0,Y 219.508,Z 730.374,A -85,B 0,C 180,E1 -25224.152,E2 -25224.152} C_VEL
LIN {X 0,Y 213.762,Z 745.903,A -85,B 0,C 180,E1 -25225.24,E2 -25225.24} C_VEL
LIN {X 0,Y 208.661,Z 757.712,A -85,B 0,C 180,E1 -25226.266,E2 -25226.266} C_VEL
LIN {X 0,Y 202.296,Z 770.53,A -85,B 0,C 180,E1 -25227.64,E2 -25227.64} C_VEL
LIN {X 0,Y 196.09,Z 781.656,A -85,B 0,C 180,E1 -25229.121,E2 -25229.121} C_VEL
LIN {X 0,Y 189.341,Z 792.487,A -85,B 0,C 180,E1 -25230.87,E2 -25230.87} C_VEL
LIN {X 0,Y 182.23,Z 802.941,A -85,B 0,C 180,E1 -25232.986,E2 -25232.986} C_VEL
LIN {X 0,Y 175.904,Z 811.365,A -85,B 0,C 180,E1 -25235.012,E2 -25235.012} C_VEL
LIN {X 0,Y 168.696,Z 820.317,A -85,B 0,C 180,E1 -25237.671,E2 -25237.671} C_VEL
LIN {X 0,Y 161.415,Z 828.721,A -85,B 0,C 180,E1 -25240.776,E2 -25240.776} C_VEL
LIN {X 0,Y 154.658,Z 836.225,A -85,B 0,C 180,E1 -25244.3,E2 -25244.3} C_VEL
LIN {X 0,Y 147.93,Z 843.126,A -85,B 0,C 180,E1 -25248.309,E2 -25248.309} C_VEL
LIN {X 0,Y 143.323,Z 847.813,A -85,B 0,C 180,E1 -25251.682,E2 -25251.682} C_VEL
LIN {X 0,Y 138.432,Z 852.737,A -85,B 0,C 180,E1 -25256.052,E2 -25256.052} C_VEL
LIN {X 0,Y 133.6,Z 857.651,A -85,B 0,C 180,E1 -25261.743,E2 -25261.743} C_VEL
LIN {X 0,Y 130.01,Z 861.52,A -85,B 0,C 180,E1 -25267.766,E2 -25267.766} C_VEL
LIN {X 0,Y 127.535,Z 864.388,A -85,B 0,C 180,E1 -25274.007,E2 -25274.007} C_VEL
LIN {X 0,Y 126.841,Z 865.536,A -85,B 0,C 180,E1 -25277.195,E2 -25277.195} C_VEL
LIN {X 0,Y 126.247,Z 866.985,A -85,B 0,C 180,E1 -25283.608,E2 -25283.608} C_VEL
LIN {X 0,Y 126.421,Z 867.476,A -85,B 0,C 180,E1 -25290,E2 -25290} C_VEL
LIN {X 0,Y 126.247,Z 866.985,A -85,B 0,C 180,E1 -25296.392,E2 -25296.392} C_VEL
LIN {X 0,Y 126.838,Z 865.535,A -85,B 0,C 180,E1 -25302.805,E2 -25302.805} C_VEL
LIN {X 0,Y 128.629,Z 863.13,A -85,B 0,C 180,E1 -25309.136,E2 -25309.136} C_VEL
LIN {X 0,Y 131.664,Z 859.739,A -85,B 0,C 180,E1 -25315.278,E2 -25315.278} C_VEL
LIN {X 0,Y 135.833,Z 855.316,A -85,B 0,C 180,E1 -25321.157,E2 -25321.157} C_VEL
LIN {X 0,Y 139.152,Z 852.027,A -85,B 0,C 180,E1 -25324.647,E2 -25324.647} C_VEL
LIN {X 0,Y 140.782,Z 849.875,A -85,B 0,C 180,E1 -25326.796,E2 -25326.796} C_VEL
LIN {X 0,Y 143.547,Z 842.933,A -85,B 0,C 180,E1 -25333.336,E2 -25333.336} C_VEL
LIN {X 0,Y 145.918,Z 839.874,A -85,B 0,C 180,E1 -25335.585,E2 -25335.585} C_VEL
LIN {X 0,Y 146.39,Z 839.356,A -85,B 0,C 180,E1 -25335.871,E2 -25335.871} C_VEL
LIN {X 0,Y 155.084,Z 830.41,A -85,B 0,C 180,E1 -25340.388,E2 -25340.388} C_VEL
LIN {X 0,Y 161.983,Z 822.86,A -85,B 0,C 180,E1 -25343.384,E2 -25343.384} C_VEL
LIN {X 0,Y 169.309,Z 814.281,A -85,B 0,C 180,E1 -25346.117,E2 -25346.117} C_VEL
LIN {X 0,Y 177.111,Z 804.504,A -85,B 0,C 180,E1 -25348.553,E2 -25348.553} C_VEL
LIN {X 0,Y 184.338,Z 794.388,A -85,B 0,C 180,E1 -25350.648,E2 -25350.648} C_VEL
LIN {X 0,Y 191.274,Z 783.728,A -85,B 0,C 180,E1 -25352.425,E2 -25352.425} C_VEL
LIN {X 0,Y 197.65,Z 772.927,A -85,B 0,C 180,E1 -25353.872,E2 -25353.872} C_VEL
LIN {X 0,Y 203.428,Z 761.998,A -85,B 0,C 180,E1 -25355.075,E2 -25355.075} C_VEL
LIN {X 0,Y 209.275,Z 749.309,A -85,B 0,C 180,E1 -25356.234,E2 -25356.234} C_VEL
LIN {X 0,Y 214.094,Z 737.342,A -85,B 0,C 180,E1 -25357.099,E2 -25357.099} C_VEL
LIN {X 0,Y 218.589,Z 724.144,A -85,B 0,C 180,E1 -25357.872,E2 -25357.872} C_VEL
LIN {X 0,Y 222.201,Z 711.408,A -85,B 0,C 180,E1 -25358.446,E2 -25358.446} C_VEL
LIN {X 0,Y 225.038,Z 698.807,A -85,B 0,C 180,E1 -25358.905,E2 -25358.905} C_VEL
LIN {X 0,Y 227.2,Z 685.899,A -85,B 0,C 180,E1 -25359.282,E2 -25359.282} C_VEL
LIN {X 0,Y 230.744,Z 652.886,A -85,B 0,C 180,E1 -25360.004,E2 -25360.004} C_VEL
LIN {X 0,Y 234.175,Z 617.9,A -85,B 0,C 180,E1 -25360.78,E2 -25360.78} C_VEL
LIN {X 0,Y 232.644,Z 613.587,A -85,B 0,C 180,E1 -25362.298,E2 -25362.298} C_VEL
LIN {X 0,Y 230.142,Z 608.215,A -85,B 0,C 180,E1 -25364.95,E2 -25364.95} C_VEL
LIN {X 0,Y 227.494,Z 602.817,A -85,B 0,C 180,E1 -25368.416,E2 -25368.416} C_VEL
LIN {X 0,Y 225.952,Z 599.718,A -85,B 0,C 180,E1 -25371.053,E2 -25371.053} C_VEL
LIN {X 0,Y 224.41,Z 596.207,A -85,B 0,C 180,E1 -25375.059,E2 -25375.059} C_VEL
LIN {X 0,Y 223.645,Z 595.072,A -85,B 0,C 180,E1 -25380,E2 -25380} C_VEL
LIN {X 0,Y 224.477,Z 596.423,A -85,B 0,C 180,E1 -25385.614,E2 -25385.614} C_VEL
LIN {X 0,Y 226.363,Z 600.573,A -85,B 0,C 180,E1 -25390.142,E2 -25390.142} C_VEL
LIN {X 0,Y 228.219,Z 604.45,A -85,B 0,C 180,E1 -25393.07,E2 -25393.07} C_VEL
LIN {X 0,Y 230.56,Z 608.933,A -85,B 0,C 180,E1 -25395.922,E2 -25395.922} C_VEL
LIN {X 0,Y 233.954,Z 616.464,A -85,B 0,C 180,E1 -25399.351,E2 -25399.351} C_VEL
LIN {X 0,Y 242.21,Z 633.138,A -85,B 0,C 180,E1 -25405.512,E2 -25405.512} C_VEL
LIN {X 0,Y 248.661,Z 642.362,A -85,B 0,C 180,E1 -25409.039,E2 -25409.039} C_VEL
LIN {X 0,Y 256.171,Z 650.995,A -85,B 0,C 180,E1 -25412.405,E2 -25412.405} C_VEL
LIN {X 0,Y 272.573,Z 665.737,A -85,B 0,C 180,E1 -25418.148,E2 -25418.148} C_VEL
LIN {X 0,Y 283.725,Z 674.258,A -85,B 0,C 180,E1 -25421.38,E2 -25421.38} C_VEL
LIN {X 0,Y 291.577,Z 680.377,A -85,B 0,C 180,E1 -25423.833,E2 -25423.833} C_VEL
LIN {X 0,Y 297.936,Z 685.395,A -85,B 0,C 180,E1 -25426.013,E2 -25426.013} C_VEL
LIN {X 0,Y 304.614,Z 690.542,A -85,B 0,C 180,E1 -25428.465,E2 -25428.465} C_VEL
LIN {X 0,Y 311.36,Z 696.068,A -85,B 0,C 180,E1 -25431.125,E2 -25431.125} C_VEL
LIN {X 0,Y 317.304,Z 700.604,A -85,B 0,C 180,E1 -25433.592,E2 -25433.592} C_VEL
LIN {X 0,Y 323.297,Z 705.295,A -85,B 0,C 180,E1 -25436.226,E2 -25436.226} C_VEL
LIN {X 0,Y 327.518,Z 708.503,A -85,B 0,C 180,E1 -25438.176,E2 -25438.176} C_VEL
LIN {X 0,Y 332.75,Z 712.704,A -85,B 0,C 180,E1 -25440.751,E2 -25440.751} C_VEL
